// TwinCAT 3 PLC project DAS_CoreSys
// Title: DAS_TaiXin
// Company: Jidain
// ProjectVersion: 1.0.1
// ProgramVersion: 3.1.4026.20
// libraries:
//   AxisInterface_Type03, * (Beckhoff Automation)
//   BATW_Base, * (Beckhoff Automation)
//   Common Behaviour Model, * (3S - Smart Software Solutions GmbH)
//   Tc2_EtherCAT, * (Beckhoff Automation GmbH)
//   Tc2_Math, * (Beckhoff Automation GmbH)
//   Tc2_ModbusRTU, * (Beckhoff Automation GmbH)
//   Tc2_SerialCom, * (Beckhoff Automation GmbH)
//   Tc2_Standard, * (Beckhoff Automation GmbH)
//   Tc2_System, * (Beckhoff Automation GmbH)
//   Tc2_Utilities, * (Beckhoff Automation GmbH)
//   Tc3_JsonXml, * (Beckhoff Automation GmbH)
//   Tc3_MC2_AdvancedHoming, * (Beckhoff Automation GmbH)
//   Tc3_Module, * (Beckhoff Automation GmbH)
//   Tc3_PackML_V2, * (Beckhoff Automation GmbH)
//   Util, * (System)
// project tree:
//   / CoreSys.TcTTO (not stored), ModbusTask.TcTTO, MotionSync.TcTTO (not stored)
//   Library/00_PackML/01_ObjectBase/ eModeChangeState.TcDUT (not stored), FB_ModeBase_V1.TcPOU (not stored), FB_ModeBase_V2.TcPOU, I_ErrorElement.TcIO (not stored), I_ErrorSubject.TcIO (not stored)
//   Library/00_PackML/02_Mode/ E_Severity.TcDUT (not stored), E_UnitMode.TcDUT
//   Library/10_Machine/00_BaseFBs/01_FB_ObjectBase/DUTs/ E_MethodStatus_Basic.TcDUT (not stored), ST_CmdContent.TcDUT (not stored), ST_MsgContent.TcDUT (not stored)
//   Library/10_Machine/00_BaseFBs/01_FB_ObjectBase/ FB_ObjectBase.TcPOU (not stored), FB_ObjectBase_V2.TcPOU
//   Library/10_Machine/00_BaseFBs/01_FB_ObjectBase/GVLs/ Para_ObjectBase.TcGVL (not stored)
//   Library/10_Machine/00_BaseFBs/01_FB_ObjectBase/ITFs/ IBasicElement.TcIO (not stored)
//   Library/10_Machine/11_IOData/ GVL_EIP.TcGVL (not stored), GVL_Input.TcGVL (not stored), GVL_Output.TcGVL (not stored)
//   Library/10_Machine/12_MachineControl/DUTs/ AxisNo.TcDUT (not stored), E_DataFrom.TcDUT (not stored), ST_ChangeIntoProduction.TcDUT (not stored), ST_CylinderMonitor.TcDUT (not stored), ST_MotorMonitor.TcDUT (not stored), ST_TableMoveCtrl.TcDUT (not stored), ST_TableMoveService.TcDUT (not stored), ST_TableMoveStatus.TcDUT (not stored), UnitNo.TcDUT (not stored)
//   Library/10_Machine/12_MachineControl/DUTs/Cylinders/ ST_CylinderList.TcDUT, UNI_CylinderList.TcDUT (not stored)
//   Library/10_Machine/12_MachineControl/DUTs/FanucRobot/ ST_FanucRobotList.TcDUT, UNI_FanucRobotList.TcDUT
//   Library/10_Machine/12_MachineControl/DUTs/Motor/ ST_MotorList.TcDUT (not stored), UNI_MotorList.TcDUT (not stored), ST_SameSizeCVRequest.TcDUT
//   Library/10_Machine/12_MachineControl/DUTs/Service/ ST_ServiceCtrl_Base.TcDUT (not stored), ST_ServiceStatus_Base.TcDUT (not stored)
//   Library/10_Machine/12_MachineControl/DUTs/Setup/ E_ClipNo.TcDUT (not stored), ST_AllocateRobotCoordinate.TcDUT (not stored), ST_AllocateRobotPositionTable.TcDUT (not stored), ST_AxisPara.TcDUT, ST_AxisPara_Auto.TcDUT (not stored), ST_AxisPara_HalfAuto.TcDUT (not stored), ST_AxisPara_Homing.TcDUT (not stored), ST_AxisPara_Manual.TcDUT (not stored), ST_CylinderPara.TcDUT (not stored), ST_FanucRobotCCDSetting.TcDUT (not stored), ST_OutRobotCoordinate.TcDUT (not stored), ST_OutRobotPositionTable.TcDUT (not stored), ST_PositionTable.TcDUT, ST_SetupAxis.TcDUT, ST_SetupCylinder.TcDUT (not stored), ST_SetupFanucRobot.TcDUT, ST_SetupMotor.TcDUT, ST_SetupPara.TcDUT, ST_Setup_Light.TcDUT, ST_Setup_Mechanical.TcDUT
//   Library/10_Machine/12_MachineControl/ FB_MachineControl.TcPOU, GVL_Machine.TcGVL, GVL_Machine_Const.TcGVL
//   Library/10_Machine/12_MachineControl/Service/ FB_BuzzCtrl.TcPOU, FB_MachineHoming.TcPOU, FB_MachineModeSwitch.TcPOU
//   Library/10_Machine/13_ErrorHandling/ FB_ErrorHandler.TcPOU (not stored), FB_ErrorHandler_V2.TcPOU, GVL_ErrorCode.TcGVL
//   Library/10_Machine/18_HMI_Handshake/DUTs/Allocated/ ST_Auto_Allocated.TcDUT (not stored), ST_AXIS_HOMING.TcDUT (not stored), ST_AXIS_JOG.TcDUT (not stored), ST_AXIS_PTP.TcDUT (not stored), ST_HalfAuto_Allocated.TcDUT (not stored), ST_HMI_AllocateArea.TcDUT, ST_Manual_Allocated.TcDUT, ST_Manual_AllocatedRobot.TcDUT, ST_Manual_Axis.TcDUT, ST_Manual_OutRobot.TcDUT (not stored), ST_Manual_PullOut.TcDUT, ST_Manual_RoundBelt.TcDUT, ST_Manual_TransCV.TcDUT, ST_Manual_TurnTable.TcDUT (not stored)
//   Library/10_Machine/18_HMI_Handshake/DUTs/Component/ ST_DoubleValve.TcDUT (not stored), ST_MotorCommand.TcDUT (not stored), ST_SignleValve.TcDUT (not stored)
//   Library/10_Machine/18_HMI_Handshake/DUTs/ E_AllocationJob.TcDUT
//   Library/10_Machine/18_HMI_Handshake/DUTs/IOMonitor/ ST_HMI_IOMonitor.TcDUT, ST_InputTable_MitsubishiWithWheelHouse.TcDUT, ST_Input_IOMonitor.TcDUT (not stored), ST_Output_IOMonitor.TcDUT (not stored), ST_WheelhouseInput.TcDUT (not stored), ST_WheelhouseTour.TcDUT (not stored), ST_Wheelhouse_Layer.TcDUT (not stored), UNI_HMI_WheelHouseInput.TcDUT (not stored), UNI_HMI_WheelHouseInput2.TcDUT (not stored) (excluded from build)
//   Library/10_Machine/18_HMI_Handshake/DUTs/Shipping/ ST_Auto_Shipping.TcDUT (not stored), ST_HalfAuto_Shipping.TcDUT (not stored), ST_HMI_ShippingArea.TcDUT, ST_Manual_Shipping.TcDUT (not stored)
//   Library/10_Machine/18_HMI_Handshake/DUTs/Status/ ST_AllocateStatus.TcDUT (not stored), ST_Auto_Status.TcDUT (not stored), ST_AXES_STATUS.TcDUT, ST_MotorStatus.TcDUT (not stored), ST_SINGLEAXIS_STATUS.TcDUT (not stored), ST_CylinderStatus.TcDUT (not stored), ST_HalfAuto_Status.TcDUT (not stored), ST_HMI_MachineStatus.TcDUT, ST_Manual_Status.TcDUT (not stored), ST_ShippingStatus.TcDUT (not stored), ST_StorageStatus.TcDUT (not stored)
//   Library/10_Machine/18_HMI_Handshake/DUTs/Storage/ ST_Auto_Storage.TcDUT (not stored), ST_HalfAuto_Storage.TcDUT (not stored), ST_HMI_StorageArea.TcDUT, ST_Manual_FanucRobot.TcDUT, ST_Manual_Rack.TcDUT (not stored), ST_Manual_UpCV.TcDUT (not stored), ST_Manual_LowCV.TcDUT (not stored), ST_Manual_Storage.TcDUT (not stored)
//   Library/10_Machine/18_HMI_Handshake/ FB_HmiHandShake.TcPOU, GVL_ADS.TcGVL, GVL_HMI.TcGVL
//   Library/10_Machine/18_HMI_Handshake/OLD_DUTs/ E_FeedInToWareHouse_PlaceArea.TcDUT, ST_AutoMode_FeedInToWareHouseBox.TcDUT, ST_AutoMode_RobotSelfHoming.TcDUT, ST_AutoMode_ShippingLeftSideTransCV.TcDUT, E_ClampWork.TcDUT, E_FeedInEmptyBox_PickUpArea.TcDUT, E_FeedInEmptyBox_PlaceArea.TcDUT, E_HoleIndex_X.TcDUT, E_HoleIndex_Y.TcDUT, E_MachineMode.TcDUT, E_MachineState.TcDUT, E_PullOutConveyorAddress.TcDUT, E_PullOutConveyorCommandType.TcDUT, E_PullOutConveyorState.TcDUT, E_RackState.TcDUT, E_ReloadRoundBelt_PickupArea.TcDUT, E_ReloadRoundBelt_PlaceAddress.TcDUT, E_ReloadRoundBelt_PlaceArea.TcDUT, E_RobotArea.TcDUT, E_RobotClamp.TcDUT, E_RoundBeltStation.TcDUT, E_SimpleAllocateTable.TcDUT, E_WareHouse.TcDUT, E_WareHouseLayer.TcDUT, E_WareHouseSlide.TcDUT, stPositionCommand.TcDUT, st_ads_AllocateMoveStructure.TcDUT, st_ads_MachineReset.TcDUT, st_ads_OneAxisMoveWithoutPosition.TcDUT, st_ads_OneAxisMoveWithPosition.TcDUT, st_ads_OutRobtToPlateMove.TcDUT, st_ads_RobotToAllocateMove.TcDUT, ST_Alarm_Tmax.TcDUT, st_AllocateCircleMoveStructure.TcDUT, st_AllocateRobotNeedlingMove.TcDUT, ST_AllocateRobotNeedlingMoveInfo.TcDUT, st_AllocatingNeedleInfo.TcDUT, ST_AllocationJobBatchMode.TcDUT, ST_AllocationJobBatchModeInfo.TcDUT, ST_AllocationJobBatchMode_1.TcDUT, ST_AutoAddsBoxes.TcDUT, ST_AutoAddsBoxesCommand.TcDUT, ST_AutoAddsBoxesStatus.TcDUT, st_AutoMode_AllocatingJob.TcDUT, st_AutoMode_AllocatingJob_1.TcDUT, st_AutoMode_ClampingBoxesJob.TcDUT, st_AutoMode_ClampingToPlate.TcDUT, ST_AutoMode_DetectDiameter.TcDUT, ST_AutoMode_FeedInEmptyBox.TcDUT, ST_AutoMode_ReloadRoundBeltBox.TcDUT, ST_AutoMode_RobotRegionMove.TcDUT, ST_AutoMode_ShippingLeftSideTransCVFeedBack.TcDUT, ST_AutoMode_ShippingLeftSideTransCVInfo.TcDUT, ST_AutoMode_ShippingRightSideTransCV.TcDUT, ST_AutoMode_SimpleAllocateHandShake.TcDUT, st_AutoMode_SingleStepWithInterventionRequest.TcDUT, ST_AutoMode_TransCVCamera.TcDUT, ST_AutoMode_WareHouseInnerPickToRoundBelt.TcDUT, E_ShippingPlateIndex.TcDUT, E_ShippingPlateSide.TcDUT, ST_ShippingPlateToConveyor.TcDUT, ST_AutoPullOutConveyor.TcDUT, ST_AutoPullOutConveyorCommand.TcDUT, ST_AutoPullOutConveyorSatus.TcDUT, ST_AutoServoPara.TcDUT, st_AutoSixAxisAbsMoveParameter.TcDUT, st_AutoSixAxisWarehouseParameter.TcDUT, st_AutoSperate.TcDUT, ST_Auto_LowerFeedInConveyor.TcDUT, ST_Auto_LowerFeedInConveyorCommand.TcDUT, ST_Auto_LowerFeedInConveyorStatus.TcDUT, ST_Auto_UpperFeedInConveyor.TcDUT, ST_Auto_UpperFeedInConveyorCommand.TcDUT, ST_Auto_UpperFeedInConveyorFeedback.TcDUT, ST_Auto_UpperFeedInConveyorInfo.TcDUT, ST_Auto_UpperFeedInConveyorStatus.TcDUT, st_AxisControl.TcDUT, ST_BuzzCtrl.TcDUT, ST_ClampActionRecord.TcDUT, st_ClampingBoxesInfo.TcDUT, ST_ClampSetting.TcDUT, ST_ClampSetting_FeedInToWareHouse.TcDUT, ST_ClampSetting_ReloadRoundBelt.TcDUT, ST_CommandBasic.TcDUT, ST_DetectDiameterCommand.TcDUT, ST_DetectDiameterInfo.TcDUT, ST_DetectDiameterStatus.TcDUT, ST_FanucRobotGeneralCtrl.TcDUT, ST_FanucRobotReadAllOffssetDate.TcDUT, ST_FanucRobotReadSingleOffsetData.TcDUT, ST_FanucRobotWriteAllOffsetDate.TcDUT, ST_FanucRobotWriteSingleOffsetData.TcDUT, ST_FanucRobot_CSharpCommand.TcDUT, ST_FanucRobot_CSharpStatus.TcDUT, ST_FeedInEmptyBox_Ctrl.TcDUT, ST_FeedInEmptyBox_Info.TcDUT, ST_FeedInEmptyBox_Status.TcDUT, ST_FeedInRBActionRecord.TcDUT, ST_FeedInRBBatch.TcDUT, ST_FeedInRBFlowInfo.TcDUT, ST_FeedInToWareHouseBox_Info.TcDUT, ST_FeedInToWareHouse_Ctrl.TcDUT, ST_FeedInToWareHouse_Status.TcDUT, st_FlowBaseCore.TcDUT, st_HandshakeBase.TcDUT, st_HandShakeBaseWithError.TcDUT, st_ListRunCore.TcDUT, ST_ManualServoPara.TcDUT, ST_MechanicalList.TcDUT, st_ModbusSwitchOff.TcDUT, ST_Mode.TcDUT, st_MoveConveyorJob.TcDUT, ST_OffsetData.TcDUT, st_OneDirectionCore.TcDUT, ST_OneProcessServoPara.TcDUT, ST_OpPannelStatus.TcDUT, st_OutRobotParameterCore.TcDUT, ST_PositionOffsetData.TcDUT, ST_PullOutConveyorInfo.TcDUT, ST_ReadAllOffsetDataCommand.TcDUT, ST_ReadAllOffsetDateStatus.TcDUT, ST_ReadSingleOffsetData_Command.TcDUT, ST_ReadSingleOffsetData_Info.TcDUT, ST_ReadSingleOffsetData_Status.TcDUT, st_RegionHome.TcDUT (not stored), ST_ReloadRoundBeltBox_Info.TcDUT, ST_ReloadRoundBelt_Ctrl.TcDUT, ST_ReloadRoundBelt_Status.TcDUT, st_Robot.TcDUT, st_RobotMoveAbs.TcDUT, ST_RobotRegionMove_Info.TcDUT, ST_RoundBeltCoordinates.TcDUT, st_SafetyByPass.TcDUT, ST_SaveParaDefault.TcDUT, ST_SaveParaRemote.TcDUT, st_ServiceTimeoutSetting.TcDUT, ST_ServoList.TcDUT, ST_ServoParaBasic.TcDUT, ST_SimpleAllocateCommand.TcDUT, ST_SimpleAllocateInfo.TcDUT, ST_SimpleAllocateStatus.TcDUT, st_SixAxisRobotCore.TcDUT, st_SixAxisWarehouseParameter.TcDUT, st_StationPositions.TcDUT, ST_StatusBasic.TcDUT, ST_SystemParameter.TcDUT, ST_WareHouseCoordinates.TcDUT, ST_WareHouseInnerPickBatch.TcDUT, ST_WareHouseInnerPickFlowInfo.TcDUT, ST_WriteAllOffsetData_Command.TcDUT, ST_WriteAllOffsetData_Info.TcDUT, ST_WriteAllOffsetData_Status.TcDUT, ST_WriteSingleOffsetData_Command.TcDUT, ST_WriteSingleOffsetData_Info.TcDUT, ST_WriteSingleOffsetData_Status.TcDUT
//   Library/10_Machine/18_HMI_Handshake/OLD_DUTs/DataCore/ st_ADSBaseParaCore.TcDUT (not stored), st_ADSMotoCore.TcDUT (not stored), st_ADSMotoMoveCore.TcDUT (not stored), st_ADS_X.TcDUT, st_ADS_Y.TcDUT, st_AllocateParameterCore.TcDUT (not stored), st_DASCalibrationData.TcDUT (not stored)
//   Library/10_Machine/18_HMI_Handshake/Service/DUTs/AllocateBatchMode/ st_AllocateMoveAutoBatchMode_Ctrl.TcDUT (not stored), st_AllocateMoveAutoBatchMode_Status.TcDUT (not stored), st_Coordinate.TcDUT (not stored), ST_Cylinders.TcDUT (not stored), st_RoundBeltAutoSingleMove_Ctrl.TcDUT (not stored), U_Cylinders.TcDUT (not stored)
//   Library/10_Machine/18_HMI_Handshake/Service/DUTs/ ST_HMI_Handshake.TcDUT
//   Library/10_Machine/19_Device/EL1889/ ST_EbusDI16.TcDUT (not stored), ST_EbusInputModule.TcDUT (not stored), ST_InputTable.TcDUT, ST_InputTable_Mitsubishi.TcDUT (not stored), uni_InputModule.TcDUT (not stored)
//   Library/10_Machine/19_Device/EL2889/ ST_EbusDO16.TcDUT (not stored), ST_EbusOutputModule.TcDUT (not stored), ST_OutputTable.TcDUT, ST_OutputTable_Mitsubishi.TcDUT, uni_OutputModule.TcDUT
//   Library/10_Machine/19_Device/FanucRobot/DUTs/ E_ClampAction.TcDUT (not stored), E_FanucRobotOpMode.TcDUT (not stored), E_PullOutConveyorPosition.TcDUT (not stored), E_RobotAddress.TcDUT (not stored), ST_AutoMode_ShippingRobotTransfer.TcDUT, ST_AutoMode_ShippingRobot_MoveAbs.TcDUT, ST_CCD_ZoneUse.TcDUT (not stored), ST_FanucUI1.TcDUT (not stored), ST_FanucUO1.TcDUT (not stored), ST_Fanuc_AbsMove.TcDUT (not stored), ST_Fanuc_GeneralCommand.TcDUT (not stored), ST_Fanuc_GeneralCommand_1.TcDUT (not stored), ST_Fanuc_Status.TcDUT (not stored), ST_Fanuc_WarehouseHandshake.TcDUT (not stored), ST_IntToBool.TcDUT (not stored), ST_ReadWriteParaCmd.TcDUT (not stored), ST_ReadWriteParaStatus.TcDUT
//   Library/10_Machine/19_Device/FanucRobot/ FB_FanucRobot_Basic.TcPOU (excluded from build), FB_FanucRobot_Basic_V2.TcPOU (unreadable)
//   Library/20_MachineUnits/21_StorageArea/210_Cabinet/DUTs/ E_CabinetJob.TcDUT (not stored), st_LayerStatus.TcDUT (not stored), st_WarehouseLayer.TcDUT (not stored), st_WarehouseList.TcDUT (not stored), U_Bits_To_stStatus.TcDUT (not stored), _st_LayerStatus.TcDUT (not stored), _st_WareHouseLayer.TcDUT (not stored), _st_WarehouseList.TcDUT (not stored)
//   Library/20_MachineUnits/21_StorageArea/210_Cabinet/ FB_WareHouse.TcPOU
//   Library/20_MachineUnits/21_StorageArea/210_Cabinet/Services/ FB_FeedInBox.TcPOU, FB_ReloadBox.TcPOU
//   Library/20_MachineUnits/21_StorageArea/Duts/ E_FeedInAction.TcDUT (not stored), E_FeedInToWareHouseAction.TcDUT, E_ReloadRoundBoxAction.TcDUT (not stored), st_RebootModbusDevices.TcDUT, st_RobotAbsMove_Ctrl.TcDUT (not stored), st_RobotAbsMove_Status.TcDUT (not stored), st_RobotWarehouseMove_Ctrl.TcDUT (not stored), st_RobotWarehouseMove_Status.TcDUT (not stored), ST_StorageService.TcDUT
//   Library/20_MachineUnits/21_StorageArea/ FB_StorageArea.TcPOU
//   Library/20_MachineUnits/21_StorageArea/Old_version_Service/ FB_FeedInEmptyBoxWithRobot.TcPOU (excluded from build), FB_FeedInEmptyBoxWithRobot_V2.TcPOU (not stored) (excluded from build), FB_FeedInEmptyBoxWithRobot_V3.TcPOU, FB_FeedInRoundBeltBoxBatch_Old.TcPOU (excluded from build), FB_FeedInRoundBeltBoxToWareHouse_Old.TcPOU (excluded from build), FB_FeedInRoundBeltBoxToWareHouse_OldV2.TcPOU (excluded from build), FB_ReloadRoundBeltBoxWithRobot.TcPOU (not stored) (excluded from build), FB_RobotAbsMove.TcPOU (excluded from build), FB_RobotRegionMove_FeedInConveyor.TcPOU (excluded from build), FB_WareHouseInnerPickToRoundBeltBatch_Old.TcPOU (excluded from build), FB_WareHouseWithRobotMove.TcPOU (not stored) (excluded from build)
//   Library/20_MachineUnits/21_StorageArea/Service/ FB_AddBoxes_v2.TcPOU, FB_BoxSupplyCtrl.TcPOU, FB_BoxSupplyCtrl_v1.TcPOU, FB_DiameterMovement.TcPOU, FB_LowerFeedInConveyor.TcPOU, FB_RebootModbusDevice.TcPOU, FB_StorageHoming.TcPOU, FB_UpperFeedInConveyor.TcPOU
//   Library/20_MachineUnits/21_StorageArea/Service_Robot/ FB_FeedInEmptyBoxWithRobot_V4.TcPOU, FB_FeedInRoundBeltBoxBatch.TcPOU, FB_FeedInRoundBeltBoxToWareHouse.TcPOU, FB_ReloadRoundBeltBoxWithRobot_V2.TcPOU, FB_RobotAbsMove_V2.TcPOU, FB_RobotRegionMove_AllocatedConveyor.TcPOU, FB_RobotRegionMove_BufferArea.TcPOU, FB_RobotRegionMove_FeedInConveyor_V2.TcPOU, FB_RobotRegionMove_PullOutConveyor.TcPOU, FB_RobotRegionMove_RoundBelt.TcPOU, FB_RobotSelfHoming.TcPOU, FB_WareHouseInnerPickToRoundBelt.TcPOU, FB_WareHouseInnerPickToRoundBeltBatch.TcPOU, FB_WareHouseWithRobotMove_V3.TcPOU
//   Library/20_MachineUnits/22_AllocateArea/Duts/Enums/ E_RoundBeltControlAccess.TcDUT (not stored)
//   Library/20_MachineUnits/22_AllocateArea/Duts/ E_Pistons.TcDUT (not stored), F_Even.TcPOU (not stored), ST_AllocateService.TcDUT, ST_AutoMode_ReverseBatchPick.TcDUT, E_ReverseBoxDestination.TcDUT, ST_AutoMode_ReverseBoxToWareHouse.TcDUT, ST_DuoCylinders.TcDUT (not stored), ST_ReverseBatchBoxQueue.TcDUT, ST_ReverseBatchBoxResult.TcDUT, st_RoundBeltAutoSingleMove_Status.TcDUT (not stored), Uni_DuoCylinders.TcDUT (not stored)
//   Library/20_MachineUnits/22_AllocateArea/ FB_AllocateAreaWithRoundbelt.TcPOU, FB_AllocateAreaWithXPlanar.TcPOU (not stored)
//   Library/20_MachineUnits/22_AllocateArea/FUNs/ FUN_GetNeedleCoordinates.TcPOU (not stored), FUN_GetSyncGroup_AllocationJob.TcPOU (not stored)
//   Library/20_MachineUnits/22_AllocateArea/Old_Version_Service/ FB_AllocateMoveAutoBatchMode_Reverse_Old.TcPOU (excluded from build), FB_OutRobot_BoxMoveReverse_Old.TcPOU (excluded from build), FB_OutRobot_EmptyBoxMove_old.TcPOU (excluded from build), FB_OutRobot_RareBoxMove_old.TcPOU (excluded from build), FB_PullOutConveyorAction_OLD.TcPOU (excluded from build), FB_PullOutConveyorBtnCtrl_OLD.TcPOU (excluded from build)
//   Library/20_MachineUnits/22_AllocateArea/Service/ FB_AllocateMoveAutoBatchMode_Reverse.TcPOU, FB_AllocateRobotNeedlingMove.TcPOU, FB_AllocateMoveAutoBatchMode.TcPOU, FB_OutRobot_BoxMoveReverse.TcPOU, FB_OutRobot_EmptyBoxMove.TcPOU, FB_OutRobot_BoxMoveTurnTableToRoundBelt.TcPOU, FB_OutRobot_RareBoxMove.TcPOU, FB_PullOutConveyorAction.TcPOU, FB_PullOutConveyorBtnCtrl.TcPOU (not stored), FB_RoundBeltService.TcPOU, FB_AllocateAreaHome.TcPOU, FB_SameSizeCVCamera.TcPOU, FB_DifferentCVCamera.TcPOU, FB_SameSizeCVCamera_Reverse.TcPOU, FB_SameSizeCV_ReverseBatchPickAndPhoto.TcPOU, FB_SameSizeCV_ReverseBoxToWareHouse.TcPOU, FB_TurnTableService.TcPOU
//   Library/20_MachineUnits/23_ShippingArea/Duts/ ST_BlinkInfo.TcDUT, ST_ShippingRobotTransfer_AreaInfo.TcDUT, ST_ShippingRobotTransfer_Info.TcDUT, ST_ShippingService.TcDUT
//   Library/20_MachineUnits/23_ShippingArea/ FB_ShippingArea.TcPOU, FB_ShippingHoming.TcPOU
//   Library/20_MachineUnits/23_ShippingArea/RobotService/ FB_ShippingRobotTransfer.TcPOU, FB_ShippingRobot_Buffer.TcPOU, FB_ShippingPlateScan.TcPOU, FB_ShippingRobot_Left.TcPOU, FB_ShippingRobot_PhotoStandByPos.TcPOU, FB_ShippingRobot_Right.TcPOU, FB_ShippingRobot_TransmitCVEnd.TcPOU
//   Library/20_MachineUnits/23_ShippingArea/Service/ FB_ShippingTransCV_LeftSide.TcPOU, FB_ShippingTransCV_RightSide.TcPOU
//   Library/99_Utilities/Duts/ E_SignalTowerLampMode.TcDUT (not stored), ST_BoolList.TcDUT (not stored), ST_SignalTower.TcDUT (not stored), uni_IntToBool.TcDUT (not stored)
//   Library/99_Utilities/ErrorHandling/ FB_ErrorHandler_OLD.TcPOU (not stored) (excluded from build), FB_ErrorHandler_abond.TcPOU (not stored) (excluded from build), FB_ErrorHandling.TcPOU (not stored) (excluded from build)
//   Library/99_Utilities/ FB_CylinderManualCtrl.TcPOU, FB_EdgeDetect.TcPOU (not stored), FB_MotorManualCtrl.TcPOU, FB_SignalGen.TcPOU (not stored), FB_SignalTower.TcPOU, FB_TableMove.TcPOU, FB_XY_Move.TcPOU (not stored), FB_XY_PickAndPlace.TcPOU (not stored), F_FtoPT.TcPOU (not stored)
//   Library/99_Utilities/FUNCTION/ FUN_CheckAxisAllowMove.TcPOU (not stored), FUN_CheckInPos.TcPOU, FUN_GetPositionTableData.TcPOU (not stored), FUN_MachineState.TcPOU (not stored), FUN_ResetStorageCylinder.TcPOU (not stored), FUN_RetractStorageCylinder.TcPOU (not stored)
//   Library/30_Simulation/ GVL_SimMode.TcGVL
//   Library/30_Simulation/10_IOSim/ FB_SimulatedIO.TcPOU
//   POUs/CheckProg/ CheckBounds.TcPOU (not stored), CheckDivDInt.TcPOU (not stored), CheckDivLInt.TcPOU (not stored), CheckDivLReal.TcPOU (not stored), CheckDivReal.TcPOU (not stored), CheckLRangeSigned.TcPOU (not stored), CheckLRangeUnsigned.TcPOU (not stored), CheckPointer.TcPOU (not stored), CheckRangeSigned.TcPOU (not stored), CheckRangeUnsigned.TcPOU (not stored)
//   POUs/ DAS_CoreSys.TcPOU, DAS_MotionSync.TcPOU (not stored)
//   POUs/ModbusRTU/00_BaseFBs/01_FB_ObjectBase/ FB_ObjectBase_V2.TcPOU (not stored)
//   POUs/ModbusRTU/ ComModbusRTU.TcPOU
//   POUs/ModbusRTU/SerialComTask/DUTs/ un_RS485States.TcDUT (not stored), un_RS485States_all.TcDUT (not stored)
//   POUs/ModbusRTU/SerialComTask/ FB_CommunicateModbusRTU.TcPOU
//   POUs/RS485_JidianVersion/DUTs/ ST_RS485Controller.TcDUT, ST_RS485_Heartbeat.TcDUT, ST_RS485_LayerStatus.TcDUT, ST_RS485_SliderStatusALL.TcDUT
//   POUs/RS485_JidianVersion/ FB_WarehouseSensorCtrl.TcPOU, MAIN2_RS485.TcPOU
// real-time tasks:
//   TASK CoreSys: cycle T#10ms, priority 20, ADS port 350
//   TASK MotionSync: cycle T#2ms, priority 1, ADS port 351
//   TASK EIP_Task: cycle T#2ms, priority 2, ADS port 301
//   TASK ModbusTask: cycle T#5ms, priority 21, ADS port 352
// motion (NC):
//   TASK NC-Task 1 SAF: cycle T#2ms, priority 4, ADS port 501
//   TASK NC-Task 1 SVB: cycle T#2ms, priority 8, ADS port 511
//   AXIS Axis 1|TurnTable (id 1)
//     General: UnitName=°
//     Dynamic: Acceleration=1800, Deceleration=1800, Jerk=10800
//     Velo: SlowManual=6, FastManual=60, Maximum=600
//     OtherSettings: AllowMotionCmdToSlave=true
//     encoder EncType=19
//       EncPara: ScaleFactorNumerator=120, ScaleFactorDenominator=83886080, MaxCount=#xffffffff
//         SoftEndMaxControl: Range=350
//         Inc: RefSoftSyncMask=#x0000ffff
//     drive DrvType=16
//       DrvPara: MaxCount=#xffffffff, DriveControlDWord=#x00020100
//         Analog: VeloReferenz=600, TorqueSetpointScale=10, ScaleFactorActTorque=0.1
//         TimeComp: TaskDelayCycles=1
//     controller CtrType=1
//       CtrPara: PriorControlFactor=1
//         PosDiffControl: Enable=false
//         Observer: BandWidth=20
//   AXIS Axis 2|RoundBelt (id 2)
//     General: UnitFlags=#x00000004
//     Dynamic: AccelerationMaximum=3900, DecelerationMaximum=3900, Acceleration=3900, Deceleration=3900, Jerk=30000
//     Velo: SlowManual=6, FastManual=200, Maximum=500
//     OtherSettings: AllowMotionCmdToSlave=true
//     encoder EncType=19
//       EncPara: ScaleFactorNumerator=500, ScaleFactorDenominator=167772160, ModuloFactor=2800, MaxCount=#xffffffff
//         Inc: RefSoftSyncMask=#x0000ffff
//     drive DrvType=16
//       DrvPara: MaxCount=#xffffffff, DriveControlDWord=#x00020100
//         Analog: VeloReferenz=500, TorqueSetpointScale=10, ScaleFactorActTorque=0.1
//         TimeComp: TaskDelayCycles=1
//     controller CtrType=1
//       CtrPara: PriorControlFactor=1
//         PosDiffControl: Range=10
//         Observer: BandWidth=20
//   AXIS Axis 3|AllocateRobot_X (id 3)
//     Dynamic: Acceleration=12000, Deceleration=12000, Jerk=360000
//     Velo: SlowManual=6, FastManual=60, Maximum=800
//     OtherSettings: AllowMotionCmdToSlave=true
//     encoder EncType=19
//       EncPara: ScaleFactorNumerator=36, ScaleFactorDenominator=8388608, MaxCount=#xffffffff
//         Inc: RefSoftSyncMask=#x0000ffff
//     drive DrvType=16
//       DrvPara: MaxCount=#xffffffff, DriveControlDWord=#x00020100
//         Analog: TorqueSetpointScale=10, ScaleFactorActTorque=0.1
//         TimeComp: TaskDelayCycles=1
//     controller CtrType=1
//       CtrPara: PriorControlFactor=1
//         Observer: BandWidth=20
//   AXIS Axis 4|AllocateRobot_Y (id 4)
//     Dynamic: Acceleration=15000, Deceleration=15000, Jerk=225000
//     OtherSettings: AllowMotionCmdToSlave=true
//     encoder EncType=19
//       EncPara: ScaleFactorNumerator=16, ScaleFactorDenominator=8388608, Inverse=true, MaxCount=#xffffffff
//         Inc: RefSoftSyncMask=#x0000ffff
//     drive DrvType=16
//       DrvPara: Inverse=true, MaxCount=#xffffffff, DriveControlDWord=#x00020100
//         Analog: TorqueSetpointScale=10, ScaleFactorActTorque=0.1
//         TimeComp: TaskDelayCycles=1
//     controller CtrType=1
//       CtrPara: PriorControlFactor=1
//         PosDiffControl: Range=10
//         Observer: BandWidth=20
//   AXIS Axis 5|OutRobot_X (id 5)
//     Dynamic: Acceleration=11250, Deceleration=11250, Jerk=168750
//     Velo: SlowManual=6, FastManual=60, Maximum=1500
//     OtherSettings: AllowMotionCmdToSlave=true
//     encoder EncType=19
//       EncPara: ScaleFactorNumerator=30, ScaleFactorDenominator=8388608, MaxCount=#xffffffff
//     drive DrvType=16
//       DrvPara: MaxCount=#xffffffff, DriveControlDWord=#x00020100
//         Analog: TorqueSetpointScale=10, ScaleFactorActTorque=0.1
//         TimeComp: TaskDelayCycles=1
//     controller CtrType=1
//       CtrPara: PriorControlFactor=1
//         PosDiffControl: Range=10
//         Observer: BandWidth=20
//   AXIS Axis 6|OutRobot_Y (id 6)
//     Dynamic: Acceleration=6000, Deceleration=6000, Jerk=36000
//     Velo: SlowManual=6, FastManual=60
//     OtherSettings: AllowMotionCmdToSlave=true
//     encoder EncType=19
//       EncPara: ScaleFactorNumerator=40, ScaleFactorDenominator=8388608, MaxCount=#xffffffff
//     drive DrvType=16
//       DrvPara: MaxCount=#xffffffff, DriveControlDWord=#x00020100
//         Analog: TorqueSetpointScale=10, ScaleFactorActTorque=0.1
//         TimeComp: TaskDelayCycles=1
//     controller CtrType=1
//       CtrPara: PriorControlFactor=1
//         PosDiffControl: Range=10
//         Observer: BandWidth=20
//   AXIS Axis 7|RackMotor (id 7)
//     Dynamic: Acceleration=800.624, Deceleration=800.624, Jerk=1167.58
//     Velo: SlowManual=5, FastManual=100, Maximum=732
//     OtherSettings: AllowMotionCmdToSlave=true
//     encoder EncType=4
//       EncPara: ScaleFactorNumerator=90, ScaleFactorDenominator=980, MaxCount=#xffffffff
//     drive DrvType=23
//       Analog: VeloReferenz=732, TorqueSetpointScale=10, ScaleFactorActTorque=0.1
//       TimeComp: TaskDelayCycles=1
//     controller CtrType=1
//       CtrPara: PriorControlFactor=1
//         PID: PosKp=90
//         Observer: BandWidth=20
// I/O:
//   DEVICE Device 1 (EtherCAT) Storage, AmsNetId 169.254.53.69.2.1
//     Term 1 (EK1200) [EK1200-5000 EtherCAT Power supply (2A E-Bus)]
//       Term 2 (EL6021) [EL6021 Interface (RS422/485)]
//       Term 3 (EL6021) [EL6021 Interface (RS422/485)]
//       Term 4 (EL6021) [EL6021 Interface (RS422/485)]
//       Term 5 (EL6021) [EL6021 Interface (RS422/485)]
//       Term 6 (EL1889)_01(X6) [EL1889 16Ch. Dig. Input 24V, 3ms, negative]
//       Term 7 (EL1889)_02(X7) [EL1889 16Ch. Dig. Input 24V, 3ms, negative]
//       Term 8 (EL1889)_03(X9) [EL1889 16Ch. Dig. Input 24V, 3ms, negative]
//       Term 9 (EL1889)_04(X10) [EL1889 16Ch. Dig. Input 24V, 3ms, negative]
//       Term 10 (EL2889)_01(Y4) [EL2889 16Ch. Dig. Output 24V, 0.5A, negative]
//       Term 11 (EL2889)_02(Y5) [EL2889 16Ch. Dig. Output 24V, 0.5A, negative]
//       Term 12 (EL2889)_03(Y6) [EL2889 16Ch. Dig. Output 24V, 0.5A, negative]
//       Term 13 (EL2889)_04(Y7) [EL2889 16Ch. Dig. Output 24V, 0.5A, negative]
//       Term 14 (EL2889)_05(Y8) [EL2889 16Ch. Dig. Output 24V, 0.5A, negative]
//       Term 59 (EL9410) [EL9410 E-Bus Power Supplier  (Diagnostics)]
//       Term 15 (EL2889)_06(Y10) [EL2889 16Ch. Dig. Output 24V, 0.5A, negative]
//       Term 17 (EL2889)_07(Y11) [EL2889 16Ch. Dig. Output 24V, 0.5A, negative]
//       Term 18 (EL7342) [EL7342 2Ch. DC motor output stage (50V, 3.5A)]
//       Term 19 (EL6652) [EL6652 EtherNet/IP Scanner (Master)]
//       Term 20 (EL9011) [EL9011 End Terminal]
//   DEVICE Device 4 (EtherCAT) Allocate, AmsNetId 169.254.53.69.5.1
//     Box 21 (CU2508) [CU2508 Ethernet Port]
//     Term 22 (EK1100) [EK1100 EtherCAT Coupler (2A E-Bus)]
//       Term 23 (EL1889)_05(X0) [EL1889 16Ch. Dig. Input 24V, 3ms, negative]
//       Term 24 (EL1889)_06(X1) [EL1889 16Ch. Dig. Input 24V, 3ms, negative]
//       Term 25 (EL1889)_07(X2) [EL1889 16Ch. Dig. Input 24V, 3ms, negative]
//       Term 26 (EL1889)_08(X3) [EL1889 16Ch. Dig. Input 24V, 3ms, negative]
//       Term 27 (EL1889)_09(X8) [EL1889 16Ch. Dig. Input 24V, 3ms, negative]
//       Term 28 (EL1889)_10(X11) [EL1889 16Ch. Dig. Input 24V, 3ms, negative]
//       Term 29 (EL2889)_08(Y0) [EL2889 16Ch. Dig. Output 24V, 0.5A, negative]
//       Term 30 (EL2889)_09(Y1) [EL2889 16Ch. Dig. Output 24V, 0.5A, negative]
//       Term 31 (EL2889)_10(Y2) [EL2889 16Ch. Dig. Output 24V, 0.5A, negative]
//       Term 32 (EL9410) [EL9410 E-Bus Power Supplier  (Diagnostics)]
//       Term 33 (EL1889)_11(X4) [EL1889 16Ch. Dig. Input 24V, 3ms, negative]
//       Term 15 (EL6652) [EL6652 EtherNet/IP Scanner (Master)]
//       Term 16 (EL9011) [EL9011 End Terminal]
//   DEVICE Device 5 (EtherCAT), AmsNetId 169.254.53.69.6.1
//     Box 37 (CU2508) [CU2508 Ethernet Port]
//     Drive 38 (MBDLT25BF) [MBDLT25BF]
//     Drive 39 (MCDLT35BF) [MCDLT35BF]
//     Drive 40 (MBDLT25BF) [MBDLT25BF]
//     Drive 41 (MADLT15BF) [MADLT15BF]
//     Drive 42 (MADLT15BF) [MADLT15BF]
//     Drive 43 (MBDLT25BF) [MBDLT25BF]
//   DEVICE Storage Fanuc Robot (ECAT EIP Scanner (EL6652)), AmsNetId 169.254.53.69.4.1
//     FANUC Robot R30iB+ // <INFO> 192.168.0.3, FANUC Robot R30iB+ (ProdCode: 4, Rev: 3.01, Mac: 00:e0:e4:c5:29:bd) </INFO> <EDS> C:\TwinCAT\3.1\Config\Io\EtherNetIP\FANUCROBOT0301_R30IBP.EDS </EDS>
//   DEVICE Device 6 (ECAT EIP Scanner (EL6652)), AmsNetId 169.254.53.69.7.1
//     FANUC Robot R30iB+ // <INFO> 192.168.0.13, FANUC Robot R30iB+ (ProdCode: 4, Rev: 3.01, Mac: 00:e0:e4:99:c3:31) </INFO> <EDS> C:\TwinCAT\3.1\Config\Io\EtherNetIP\FANUCROBOT0301_R30IBP.EDS </EDS>
//   DEVICE X001 (RT-Ethernet Adapter)
// variable links:
//   NC-Task 1 SAF/Axes/Axis 1|TurnTable <-> Device 5 (EtherCAT)/Drive 38 (MBDLT25BF)
//     Drive/Inputs/In/nDataIn1 <-> Transmit PDO mapping 1/Following error actual value
//     Drive/Inputs/In/nDcOutputTime <-> InfoData/DcOutputShift
//     Drive/Inputs/In/nState1 <-> Transmit PDO mapping 1/Statusword
//     Drive/Inputs/In/nState2 <-> Transmit PDO mapping 1/Statusword @bit 8
//     Drive/Inputs/In/nState4 @bit 1 <-> WcState/InputToggle
//     Drive/Inputs/In/nState4 <-> WcState/WcState
//     Drive/Inputs/In/nState5 <-> Transmit PDO mapping 1/Modes of operation display
//     Drive/Outputs/Out/nCtrl1 <-> Receive PDO mapping 1/Controlword
//     Drive/Outputs/Out/nCtrl2 <-> Receive PDO mapping 1/Controlword @bit 8
//     Drive/Outputs/Out/nCtrl5 <-> Receive PDO mapping 1/Modes of operation
//     Drive/Outputs/Out/nDataOut1 <-> Receive PDO mapping 1/Target position
//     Enc/Inputs/In/nDataIn1 <-> Transmit PDO mapping 1/Position actual value
//     Enc/Inputs/In/nDataIn3 <-> Transmit PDO mapping 1/Touch probe pos1 pos value
//     Enc/Inputs/In/nDcInputTime <-> InfoData/DcInputShift
//     Enc/Inputs/In/nState4 @bit 1 <-> WcState/InputToggle
//     Enc/Inputs/In/nState4 <-> WcState/WcState
//     Enc/Inputs/In/nState5 <-> Transmit PDO mapping 1/Touch probe status
//     Enc/Inputs/In/nState6 <-> Transmit PDO mapping 1/Touch probe status @bit 8
//     Enc/Outputs/Out/nCtrl5 <-> Receive PDO mapping 1/Touch probe function
//     Enc/Outputs/Out/nCtrl6 <-> Receive PDO mapping 1/Touch probe function @bit 8
//   NC-Task 1 SAF/Axes/Axis 2|RoundBelt <-> Device 5 (EtherCAT)/Drive 39 (MCDLT35BF)
//     Drive/Inputs/In/nDataIn1 <-> Transmit PDO mapping 1/Following error actual value
//     Drive/Inputs/In/nDataIn3[0] <-> Transmit PDO mapping 1/Torque actual value
//     Drive/Inputs/In/nDcOutputTime <-> InfoData/DcOutputShift
//     Drive/Inputs/In/nState1 <-> Transmit PDO mapping 1/Statusword
//     Drive/Inputs/In/nState2 <-> Transmit PDO mapping 1/Statusword @bit 8
//     Drive/Inputs/In/nState4 @bit 1 <-> WcState/InputToggle
//     Drive/Inputs/In/nState4 <-> WcState/WcState
//     Drive/Inputs/In/nState5 <-> Transmit PDO mapping 1/Modes of operation display
//     Drive/Outputs/Out/nCtrl1 <-> Receive PDO mapping 1/Controlword
//     Drive/Outputs/Out/nCtrl2 <-> Receive PDO mapping 1/Controlword @bit 8
//     Drive/Outputs/Out/nCtrl5 <-> Receive PDO mapping 1/Modes of operation
//     Drive/Outputs/Out/nDataOut1 <-> Receive PDO mapping 1/Target position
//     Enc/Inputs/In/nDataIn1 <-> Transmit PDO mapping 1/Position actual value
//     Enc/Inputs/In/nDataIn3 <-> Transmit PDO mapping 1/Touch probe pos1 pos value
//     Enc/Inputs/In/nDcInputTime <-> InfoData/DcInputShift
//     Enc/Inputs/In/nState4 @bit 1 <-> WcState/InputToggle
//     Enc/Inputs/In/nState4 <-> WcState/WcState
//     Enc/Inputs/In/nState5 <-> Transmit PDO mapping 1/Touch probe status
//     Enc/Inputs/In/nState6 <-> Transmit PDO mapping 1/Touch probe status @bit 8
//     Enc/Outputs/Out/nCtrl5 <-> Receive PDO mapping 1/Touch probe function
//     Enc/Outputs/Out/nCtrl6 <-> Receive PDO mapping 1/Touch probe function @bit 8
//   NC-Task 1 SAF/Axes/Axis 3|AllocateRobot_X <-> Device 5 (EtherCAT)/Drive 40 (MBDLT25BF)
//     Drive/Inputs/In/nDataIn1 <-> Transmit PDO mapping 1/Following error actual value
//     Drive/Inputs/In/nDcOutputTime <-> InfoData/DcOutputShift
//     Drive/Inputs/In/nState1 <-> Transmit PDO mapping 1/Statusword
//     Drive/Inputs/In/nState2 <-> Transmit PDO mapping 1/Statusword @bit 8
//     Drive/Inputs/In/nState4 @bit 1 <-> WcState/InputToggle
//     Drive/Inputs/In/nState4 <-> WcState/WcState
//     Drive/Inputs/In/nState5 <-> Transmit PDO mapping 1/Modes of operation display
//     Drive/Outputs/Out/nCtrl1 <-> Receive PDO mapping 1/Controlword
//     Drive/Outputs/Out/nCtrl2 <-> Receive PDO mapping 1/Controlword @bit 8
//     Drive/Outputs/Out/nCtrl5 <-> Receive PDO mapping 1/Modes of operation
//     Drive/Outputs/Out/nDataOut1 <-> Receive PDO mapping 1/Target position
//     Enc/Inputs/In/nDataIn1 <-> Transmit PDO mapping 1/Position actual value
//     Enc/Inputs/In/nDataIn3 <-> Transmit PDO mapping 1/Touch probe pos1 pos value
//     Enc/Inputs/In/nDcInputTime <-> InfoData/DcInputShift
//     Enc/Inputs/In/nState4 @bit 1 <-> WcState/InputToggle
//     Enc/Inputs/In/nState4 <-> WcState/WcState
//     Enc/Inputs/In/nState5 <-> Transmit PDO mapping 1/Touch probe status
//     Enc/Inputs/In/nState6 <-> Transmit PDO mapping 1/Touch probe status @bit 8
//     Enc/Outputs/Out/nCtrl5 <-> Receive PDO mapping 1/Touch probe function
//     Enc/Outputs/Out/nCtrl6 <-> Receive PDO mapping 1/Touch probe function @bit 8
//   NC-Task 1 SAF/Axes/Axis 4|AllocateRobot_Y <-> Device 5 (EtherCAT)/Drive 41 (MADLT15BF)
//     Drive/Inputs/In/nDataIn1 <-> Transmit PDO mapping 1/Following error actual value
//     Drive/Inputs/In/nDcOutputTime <-> InfoData/DcOutputShift
//     Drive/Inputs/In/nState1 <-> Transmit PDO mapping 1/Statusword
//     Drive/Inputs/In/nState2 <-> Transmit PDO mapping 1/Statusword @bit 8
//     Drive/Inputs/In/nState4 @bit 1 <-> WcState/InputToggle
//     Drive/Inputs/In/nState4 <-> WcState/WcState
//     Drive/Inputs/In/nState5 <-> Transmit PDO mapping 1/Modes of operation display
//     Drive/Outputs/Out/nCtrl1 <-> Receive PDO mapping 1/Controlword
//     Drive/Outputs/Out/nCtrl2 <-> Receive PDO mapping 1/Controlword @bit 8
//     Drive/Outputs/Out/nCtrl5 <-> Receive PDO mapping 1/Modes of operation
//     Drive/Outputs/Out/nDataOut1 <-> Receive PDO mapping 1/Target position
//     Enc/Inputs/In/nDataIn1 <-> Transmit PDO mapping 1/Position actual value
//     Enc/Inputs/In/nDataIn3 <-> Transmit PDO mapping 1/Touch probe pos1 pos value
//     Enc/Inputs/In/nDcInputTime <-> InfoData/DcInputShift
//     Enc/Inputs/In/nState4 @bit 1 <-> WcState/InputToggle
//     Enc/Inputs/In/nState4 <-> WcState/WcState
//     Enc/Inputs/In/nState5 <-> Transmit PDO mapping 1/Touch probe status
//     Enc/Inputs/In/nState6 <-> Transmit PDO mapping 1/Touch probe status @bit 8
//     Enc/Outputs/Out/nCtrl5 <-> Receive PDO mapping 1/Touch probe function
//     Enc/Outputs/Out/nCtrl6 <-> Receive PDO mapping 1/Touch probe function @bit 8
//   NC-Task 1 SAF/Axes/Axis 5|OutRobot_X <-> Device 5 (EtherCAT)/Drive 42 (MADLT15BF)
//     Drive/Inputs/In/nDataIn1 <-> Transmit PDO mapping 1/Following error actual value
//     Drive/Inputs/In/nDcOutputTime <-> InfoData/DcOutputShift
//     Drive/Inputs/In/nState1 <-> Transmit PDO mapping 1/Statusword
//     Drive/Inputs/In/nState2 <-> Transmit PDO mapping 1/Statusword @bit 8
//     Drive/Inputs/In/nState4 @bit 1 <-> WcState/InputToggle
//     Drive/Inputs/In/nState4 <-> WcState/WcState
//     Drive/Inputs/In/nState5 <-> Transmit PDO mapping 1/Modes of operation display
//     Drive/Outputs/Out/nCtrl1 <-> Receive PDO mapping 1/Controlword
//     Drive/Outputs/Out/nCtrl2 <-> Receive PDO mapping 1/Controlword @bit 8
//     Drive/Outputs/Out/nCtrl5 <-> Receive PDO mapping 1/Modes of operation
//     Drive/Outputs/Out/nDataOut1 <-> Receive PDO mapping 1/Target position
//     Enc/Inputs/In/nDataIn1 <-> Transmit PDO mapping 1/Position actual value
//     Enc/Inputs/In/nDataIn3 <-> Transmit PDO mapping 1/Touch probe pos1 pos value
//     Enc/Inputs/In/nDcInputTime <-> InfoData/DcInputShift
//     Enc/Inputs/In/nState4 @bit 1 <-> WcState/InputToggle
//     Enc/Inputs/In/nState4 <-> WcState/WcState
//     Enc/Inputs/In/nState5 <-> Transmit PDO mapping 1/Touch probe status
//     Enc/Inputs/In/nState6 <-> Transmit PDO mapping 1/Touch probe status @bit 8
//     Enc/Outputs/Out/nCtrl5 <-> Receive PDO mapping 1/Touch probe function
//     Enc/Outputs/Out/nCtrl6 <-> Receive PDO mapping 1/Touch probe function @bit 8
//   NC-Task 1 SAF/Axes/Axis 6|OutRobot_Y <-> Device 5 (EtherCAT)/Drive 43 (MBDLT25BF)
//     Drive/Inputs/In/nDataIn1 <-> Transmit PDO mapping 1/Following error actual value
//     Drive/Inputs/In/nDcOutputTime <-> InfoData/DcOutputShift
//     Drive/Inputs/In/nState1 <-> Transmit PDO mapping 1/Statusword
//     Drive/Inputs/In/nState2 <-> Transmit PDO mapping 1/Statusword @bit 8
//     Drive/Inputs/In/nState4 @bit 1 <-> WcState/InputToggle
//     Drive/Inputs/In/nState4 <-> WcState/WcState
//     Drive/Inputs/In/nState5 <-> Transmit PDO mapping 1/Modes of operation display
//     Drive/Outputs/Out/nCtrl1 <-> Receive PDO mapping 1/Controlword
//     Drive/Outputs/Out/nCtrl2 <-> Receive PDO mapping 1/Controlword @bit 8
//     Drive/Outputs/Out/nCtrl5 <-> Receive PDO mapping 1/Modes of operation
//     Drive/Outputs/Out/nDataOut1 <-> Receive PDO mapping 1/Target position
//     Enc/Inputs/In/nDataIn1 <-> Transmit PDO mapping 1/Position actual value
//     Enc/Inputs/In/nDataIn3 <-> Transmit PDO mapping 1/Touch probe pos1 pos value
//     Enc/Inputs/In/nDcInputTime <-> InfoData/DcInputShift
//     Enc/Inputs/In/nState4 @bit 1 <-> WcState/InputToggle
//     Enc/Inputs/In/nState4 <-> WcState/WcState
//     Enc/Inputs/In/nState5 <-> Transmit PDO mapping 1/Touch probe status
//     Enc/Inputs/In/nState6 <-> Transmit PDO mapping 1/Touch probe status @bit 8
//     Enc/Outputs/Out/nCtrl5 <-> Receive PDO mapping 1/Touch probe function
//     Enc/Outputs/Out/nCtrl6 <-> Receive PDO mapping 1/Touch probe function @bit 8
//   NC-Task 1 SAF/Axes/Axis 7|RackMotor <-> Device 1 (EtherCAT) Storage/Term 1 (EK1200)/Term 18 (EL7342)
//     Drive/Inputs/In/nState1 @bit 3 <-> DCM Status Channel 1/Status/Error
//     Drive/Inputs/In/nState1 @bit 5 <-> DCM Status Channel 1/Status/Moving negative
//     Drive/Inputs/In/nState1 @bit 4 <-> DCM Status Channel 1/Status/Moving positive
//     Drive/Inputs/In/nState1 @bit 1 <-> DCM Status Channel 1/Status/Ready
//     Drive/Inputs/In/nState1 <-> DCM Status Channel 1/Status/Ready to enable
//     Drive/Inputs/In/nState1 @bit 6 <-> DCM Status Channel 1/Status/Torque reduced
//     Drive/Inputs/In/nState1 @bit 2 <-> DCM Status Channel 1/Status/Warning
//     Drive/Inputs/In/nState2 @bit 3 <-> DCM Status Channel 1/Status/Digital input 1
//     Drive/Inputs/In/nState2 @bit 4 <-> DCM Status Channel 1/Status/Digital input 2
//     Drive/Inputs/In/nState2 @bit 5 <-> DCM Status Channel 1/Status/Sync error
//     Drive/Inputs/In/nState2 @bit 7 <-> DCM Status Channel 1/Status/TxPDO Toggle
//     Drive/Inputs/In/nState4 @bit 1 <-> WcState/InputToggle
//     Drive/Inputs/In/nState4 <-> WcState/WcState
//     Drive/Outputs/Out/nCtrl1 <-> DCM Control Channel 1/Control/Enable
//     Drive/Outputs/Out/nCtrl1 @bit 2 <-> DCM Control Channel 1/Control/Reduce torque
//     Drive/Outputs/Out/nCtrl1 @bit 1 <-> DCM Control Channel 1/Control/Reset
//     Drive/Outputs/Out/nCtrl1 @bit 3 <-> DCM Control Channel 1/Control/Threshold active
//     Drive/Outputs/Out/nDataOut2[0] <-> DCM Velocity Channel 1/Velocity
//     Enc/Inputs/In/nDataIn1 <-> ENC Status Channel 1/Counter value
//     Enc/Inputs/In/nDataIn2 <-> ENC Status Channel 1/Latch value
//     Enc/Inputs/In/nState1 @bit 4 <-> ENC Status Channel 1/Status/Counter overflow
//     Enc/Inputs/In/nState1 @bit 3 <-> ENC Status Channel 1/Status/Counter underflow
//     Enc/Inputs/In/nState1 @bit 7 <-> ENC Status Channel 1/Status/Extrapolation stall
//     Enc/Inputs/In/nState1 @bit 1 <-> ENC Status Channel 1/Status/Latch extern valid
//     Enc/Inputs/In/nState1 @bit 2 <-> ENC Status Channel 1/Status/Set counter done
//     Enc/Inputs/In/nState2 @bit 4 <-> ENC Status Channel 1/Status/Status of extern latch
//     Enc/Inputs/In/nState2 <-> ENC Status Channel 1/Status/Status of input A
//     Enc/Inputs/In/nState2 @bit 1 <-> ENC Status Channel 1/Status/Status of input B
//     Enc/Inputs/In/nState2 @bit 5 <-> ENC Status Channel 1/Status/Sync error
//     Enc/Inputs/In/nState2 @bit 7 <-> ENC Status Channel 1/Status/TxPDO Toggle
//     Enc/Inputs/In/nState4 @bit 1 <-> WcState/InputToggle
//     Enc/Inputs/In/nState4 <-> WcState/WcState
//     Enc/Outputs/Out/nCtrl1 @bit 3 <-> ENC Control Channel 1/Control/Enable latch extern on negative edge
//     Enc/Outputs/Out/nCtrl1 @bit 1 <-> ENC Control Channel 1/Control/Enable latch extern on positive edge
//     Enc/Outputs/Out/nCtrl1 @bit 2 <-> ENC Control Channel 1/Control/Set counter
//     Enc/Outputs/Out/nDataOut1 <-> ENC Control Channel 1/Set counter value
//   DAS_CoreSys/DAS_CoreSys Instance <-> Device 1 (EtherCAT) Storage/Term 1 (EK1200)/Term 10 (EL2889)_01(Y4)
//     ModbusTask Outputs/GVL_Output.uniDO.stEbusDO.EL2889_01.DO1 <-> Channel 1/Output
//     ModbusTask Outputs/GVL_Output.uniDO.stEbusDO.EL2889_01.DO10 <-> Channel 10/Output
//     ModbusTask Outputs/GVL_Output.uniDO.stEbusDO.EL2889_01.DO11 <-> Channel 11/Output
//     ModbusTask Outputs/GVL_Output.uniDO.stEbusDO.EL2889_01.DO12 <-> Channel 12/Output
//     ModbusTask Outputs/GVL_Output.uniDO.stEbusDO.EL2889_01.DO13 <-> Channel 13/Output
//     ModbusTask Outputs/GVL_Output.uniDO.stEbusDO.EL2889_01.DO14 <-> Channel 14/Output
//     ModbusTask Outputs/GVL_Output.uniDO.stEbusDO.EL2889_01.DO15 <-> Channel 15/Output
//     ModbusTask Outputs/GVL_Output.uniDO.stEbusDO.EL2889_01.DO16 <-> Channel 16/Output
//     ModbusTask Outputs/GVL_Output.uniDO.stEbusDO.EL2889_01.DO2 <-> Channel 2/Output
//     ModbusTask Outputs/GVL_Output.uniDO.stEbusDO.EL2889_01.DO3 <-> Channel 3/Output
//     ModbusTask Outputs/GVL_Output.uniDO.stEbusDO.EL2889_01.DO4 <-> Channel 4/Output
//     ModbusTask Outputs/GVL_Output.uniDO.stEbusDO.EL2889_01.DO5 <-> Channel 5/Output
//     ModbusTask Outputs/GVL_Output.uniDO.stEbusDO.EL2889_01.DO6 <-> Channel 6/Output
//     ModbusTask Outputs/GVL_Output.uniDO.stEbusDO.EL2889_01.DO7 <-> Channel 7/Output
//     ModbusTask Outputs/GVL_Output.uniDO.stEbusDO.EL2889_01.DO8 <-> Channel 8/Output
//     ModbusTask Outputs/GVL_Output.uniDO.stEbusDO.EL2889_01.DO9 <-> Channel 9/Output
//   DAS_CoreSys/DAS_CoreSys Instance <-> Device 1 (EtherCAT) Storage/Term 1 (EK1200)/Term 11 (EL2889)_02(Y5)
//     ModbusTask Outputs/GVL_Output.uniDO.stEbusDO.EL2889_02.DO1 <-> Channel 1/Output
//     ModbusTask Outputs/GVL_Output.uniDO.stEbusDO.EL2889_02.DO10 <-> Channel 10/Output
//     ModbusTask Outputs/GVL_Output.uniDO.stEbusDO.EL2889_02.DO11 <-> Channel 11/Output
//     ModbusTask Outputs/GVL_Output.uniDO.stEbusDO.EL2889_02.DO12 <-> Channel 12/Output
//     ModbusTask Outputs/GVL_Output.uniDO.stEbusDO.EL2889_02.DO13 <-> Channel 13/Output
//     ModbusTask Outputs/GVL_Output.uniDO.stEbusDO.EL2889_02.DO14 <-> Channel 14/Output
//     ModbusTask Outputs/GVL_Output.uniDO.stEbusDO.EL2889_02.DO15 <-> Channel 15/Output
//     ModbusTask Outputs/GVL_Output.uniDO.stEbusDO.EL2889_02.DO16 <-> Channel 16/Output
//     ModbusTask Outputs/GVL_Output.uniDO.stEbusDO.EL2889_02.DO2 <-> Channel 2/Output
//     ModbusTask Outputs/GVL_Output.uniDO.stEbusDO.EL2889_02.DO3 <-> Channel 3/Output
//     ModbusTask Outputs/GVL_Output.uniDO.stEbusDO.EL2889_02.DO4 <-> Channel 4/Output
//     ModbusTask Outputs/GVL_Output.uniDO.stEbusDO.EL2889_02.DO5 <-> Channel 5/Output
//     ModbusTask Outputs/GVL_Output.uniDO.stEbusDO.EL2889_02.DO6 <-> Channel 6/Output
//     ModbusTask Outputs/GVL_Output.uniDO.stEbusDO.EL2889_02.DO7 <-> Channel 7/Output
//     ModbusTask Outputs/GVL_Output.uniDO.stEbusDO.EL2889_02.DO8 <-> Channel 8/Output
//     ModbusTask Outputs/GVL_Output.uniDO.stEbusDO.EL2889_02.DO9 <-> Channel 9/Output
//   DAS_CoreSys/DAS_CoreSys Instance <-> Device 1 (EtherCAT) Storage/Term 1 (EK1200)/Term 12 (EL2889)_03(Y6)
//     ModbusTask Outputs/GVL_Output.uniDO.stEbusDO.EL2889_03.DO1 <-> Channel 1/Output
//     ModbusTask Outputs/GVL_Output.uniDO.stEbusDO.EL2889_03.DO10 <-> Channel 10/Output
//     ModbusTask Outputs/GVL_Output.uniDO.stEbusDO.EL2889_03.DO11 <-> Channel 11/Output
//     ModbusTask Outputs/GVL_Output.uniDO.stEbusDO.EL2889_03.DO12 <-> Channel 12/Output
//     ModbusTask Outputs/GVL_Output.uniDO.stEbusDO.EL2889_03.DO13 <-> Channel 13/Output
//     ModbusTask Outputs/GVL_Output.uniDO.stEbusDO.EL2889_03.DO14 <-> Channel 14/Output
//     ModbusTask Outputs/GVL_Output.uniDO.stEbusDO.EL2889_03.DO15 <-> Channel 15/Output
//     ModbusTask Outputs/GVL_Output.uniDO.stEbusDO.EL2889_03.DO16 <-> Channel 16/Output
//     ModbusTask Outputs/GVL_Output.uniDO.stEbusDO.EL2889_03.DO2 <-> Channel 2/Output
//     ModbusTask Outputs/GVL_Output.uniDO.stEbusDO.EL2889_03.DO3 <-> Channel 3/Output
//     ModbusTask Outputs/GVL_Output.uniDO.stEbusDO.EL2889_03.DO4 <-> Channel 4/Output
//     ModbusTask Outputs/GVL_Output.uniDO.stEbusDO.EL2889_03.DO5 <-> Channel 5/Output
//     ModbusTask Outputs/GVL_Output.uniDO.stEbusDO.EL2889_03.DO6 <-> Channel 6/Output
//     ModbusTask Outputs/GVL_Output.uniDO.stEbusDO.EL2889_03.DO7 <-> Channel 7/Output
//     ModbusTask Outputs/GVL_Output.uniDO.stEbusDO.EL2889_03.DO8 <-> Channel 8/Output
//     ModbusTask Outputs/GVL_Output.uniDO.stEbusDO.EL2889_03.DO9 <-> Channel 9/Output
//   DAS_CoreSys/DAS_CoreSys Instance <-> Device 1 (EtherCAT) Storage/Term 1 (EK1200)/Term 13 (EL2889)_04(Y7)
//     ModbusTask Outputs/GVL_Output.uniDO.stEbusDO.EL2889_04.DO1 <-> Channel 1/Output
//     ModbusTask Outputs/GVL_Output.uniDO.stEbusDO.EL2889_04.DO10 <-> Channel 10/Output
//     ModbusTask Outputs/GVL_Output.uniDO.stEbusDO.EL2889_04.DO11 <-> Channel 11/Output
//     ModbusTask Outputs/GVL_Output.uniDO.stEbusDO.EL2889_04.DO12 <-> Channel 12/Output
//     ModbusTask Outputs/GVL_Output.uniDO.stEbusDO.EL2889_04.DO13 <-> Channel 13/Output
//     ModbusTask Outputs/GVL_Output.uniDO.stEbusDO.EL2889_04.DO14 <-> Channel 14/Output
//     ModbusTask Outputs/GVL_Output.uniDO.stEbusDO.EL2889_04.DO15 <-> Channel 15/Output
//     ModbusTask Outputs/GVL_Output.uniDO.stEbusDO.EL2889_04.DO16 <-> Channel 16/Output
//     ModbusTask Outputs/GVL_Output.uniDO.stEbusDO.EL2889_04.DO2 <-> Channel 2/Output
//     ModbusTask Outputs/GVL_Output.uniDO.stEbusDO.EL2889_04.DO3 <-> Channel 3/Output
//     ModbusTask Outputs/GVL_Output.uniDO.stEbusDO.EL2889_04.DO4 <-> Channel 4/Output
//     ModbusTask Outputs/GVL_Output.uniDO.stEbusDO.EL2889_04.DO5 <-> Channel 5/Output
//     ModbusTask Outputs/GVL_Output.uniDO.stEbusDO.EL2889_04.DO6 <-> Channel 6/Output
//     ModbusTask Outputs/GVL_Output.uniDO.stEbusDO.EL2889_04.DO7 <-> Channel 7/Output
//     ModbusTask Outputs/GVL_Output.uniDO.stEbusDO.EL2889_04.DO8 <-> Channel 8/Output
//     ModbusTask Outputs/GVL_Output.uniDO.stEbusDO.EL2889_04.DO9 <-> Channel 9/Output
//   DAS_CoreSys/DAS_CoreSys Instance <-> Device 1 (EtherCAT) Storage/Term 1 (EK1200)/Term 14 (EL2889)_05(Y8)
//     ModbusTask Outputs/GVL_Output.uniDO.stEbusDO.EL2889_05.DO1 <-> Channel 1/Output
//     ModbusTask Outputs/GVL_Output.uniDO.stEbusDO.EL2889_05.DO10 <-> Channel 10/Output
//     ModbusTask Outputs/GVL_Output.uniDO.stEbusDO.EL2889_05.DO11 <-> Channel 11/Output
//     ModbusTask Outputs/GVL_Output.uniDO.stEbusDO.EL2889_05.DO12 <-> Channel 12/Output
//     ModbusTask Outputs/GVL_Output.uniDO.stEbusDO.EL2889_05.DO13 <-> Channel 13/Output
//     ModbusTask Outputs/GVL_Output.uniDO.stEbusDO.EL2889_05.DO14 <-> Channel 14/Output
//     ModbusTask Outputs/GVL_Output.uniDO.stEbusDO.EL2889_05.DO15 <-> Channel 15/Output
//     ModbusTask Outputs/GVL_Output.uniDO.stEbusDO.EL2889_05.DO16 <-> Channel 16/Output
//     ModbusTask Outputs/GVL_Output.uniDO.stEbusDO.EL2889_05.DO2 <-> Channel 2/Output
//     ModbusTask Outputs/GVL_Output.uniDO.stEbusDO.EL2889_05.DO3 <-> Channel 3/Output
//     ModbusTask Outputs/GVL_Output.uniDO.stEbusDO.EL2889_05.DO4 <-> Channel 4/Output
//     ModbusTask Outputs/GVL_Output.uniDO.stEbusDO.EL2889_05.DO5 <-> Channel 5/Output
//     ModbusTask Outputs/GVL_Output.uniDO.stEbusDO.EL2889_05.DO6 <-> Channel 6/Output
//     ModbusTask Outputs/GVL_Output.uniDO.stEbusDO.EL2889_05.DO7 <-> Channel 7/Output
//     ModbusTask Outputs/GVL_Output.uniDO.stEbusDO.EL2889_05.DO8 <-> Channel 8/Output
//     ModbusTask Outputs/GVL_Output.uniDO.stEbusDO.EL2889_05.DO9 <-> Channel 9/Output
//   DAS_CoreSys/DAS_CoreSys Instance <-> Device 1 (EtherCAT) Storage/Term 1 (EK1200)/Term 15 (EL2889)_06(Y10)
//     ModbusTask Outputs/GVL_Output.uniDO.stEbusDO.EL2889_06.DO1 <-> Channel 1/Output
//     ModbusTask Outputs/GVL_Output.uniDO.stEbusDO.EL2889_06.DO10 <-> Channel 10/Output
//     ModbusTask Outputs/GVL_Output.uniDO.stEbusDO.EL2889_06.DO11 <-> Channel 11/Output
//     ModbusTask Outputs/GVL_Output.uniDO.stEbusDO.EL2889_06.DO12 <-> Channel 12/Output
//     ModbusTask Outputs/GVL_Output.uniDO.stEbusDO.EL2889_06.DO13 <-> Channel 13/Output
//     ModbusTask Outputs/GVL_Output.uniDO.stEbusDO.EL2889_06.DO14 <-> Channel 14/Output
//     ModbusTask Outputs/GVL_Output.uniDO.stEbusDO.EL2889_06.DO15 <-> Channel 15/Output
//     ModbusTask Outputs/GVL_Output.uniDO.stEbusDO.EL2889_06.DO16 <-> Channel 16/Output
//     ModbusTask Outputs/GVL_Output.uniDO.stEbusDO.EL2889_06.DO2 <-> Channel 2/Output
//     ModbusTask Outputs/GVL_Output.uniDO.stEbusDO.EL2889_06.DO3 <-> Channel 3/Output
//     ModbusTask Outputs/GVL_Output.uniDO.stEbusDO.EL2889_06.DO4 <-> Channel 4/Output
//     ModbusTask Outputs/GVL_Output.uniDO.stEbusDO.EL2889_06.DO5 <-> Channel 5/Output
//     ModbusTask Outputs/GVL_Output.uniDO.stEbusDO.EL2889_06.DO6 <-> Channel 6/Output
//     ModbusTask Outputs/GVL_Output.uniDO.stEbusDO.EL2889_06.DO7 <-> Channel 7/Output
//     ModbusTask Outputs/GVL_Output.uniDO.stEbusDO.EL2889_06.DO8 <-> Channel 8/Output
//     ModbusTask Outputs/GVL_Output.uniDO.stEbusDO.EL2889_06.DO9 <-> Channel 9/Output
//   DAS_CoreSys/DAS_CoreSys Instance <-> Device 1 (EtherCAT) Storage/Term 1 (EK1200)/Term 17 (EL2889)_07(Y11)
//     ModbusTask Outputs/GVL_Output.uniDO.stEbusDO.EL2889_07.DO1 <-> Channel 1/Output
//     ModbusTask Outputs/GVL_Output.uniDO.stEbusDO.EL2889_07.DO10 <-> Channel 10/Output
//     ModbusTask Outputs/GVL_Output.uniDO.stEbusDO.EL2889_07.DO11 <-> Channel 11/Output
//     ModbusTask Outputs/GVL_Output.uniDO.stEbusDO.EL2889_07.DO12 <-> Channel 12/Output
//     ModbusTask Outputs/GVL_Output.uniDO.stEbusDO.EL2889_07.DO13 <-> Channel 13/Output
//     ModbusTask Outputs/GVL_Output.uniDO.stEbusDO.EL2889_07.DO14 <-> Channel 14/Output
//     ModbusTask Outputs/GVL_Output.uniDO.stEbusDO.EL2889_07.DO15 <-> Channel 15/Output
//     ModbusTask Outputs/GVL_Output.uniDO.stEbusDO.EL2889_07.DO16 <-> Channel 16/Output
//     ModbusTask Outputs/GVL_Output.uniDO.stEbusDO.EL2889_07.DO2 <-> Channel 2/Output
//     ModbusTask Outputs/GVL_Output.uniDO.stEbusDO.EL2889_07.DO3 <-> Channel 3/Output
//     ModbusTask Outputs/GVL_Output.uniDO.stEbusDO.EL2889_07.DO4 <-> Channel 4/Output
//     ModbusTask Outputs/GVL_Output.uniDO.stEbusDO.EL2889_07.DO5 <-> Channel 5/Output
//     ModbusTask Outputs/GVL_Output.uniDO.stEbusDO.EL2889_07.DO6 <-> Channel 6/Output
//     ModbusTask Outputs/GVL_Output.uniDO.stEbusDO.EL2889_07.DO7 <-> Channel 7/Output
//     ModbusTask Outputs/GVL_Output.uniDO.stEbusDO.EL2889_07.DO8 <-> Channel 8/Output
//     ModbusTask Outputs/GVL_Output.uniDO.stEbusDO.EL2889_07.DO9 <-> Channel 9/Output
//   DAS_CoreSys/DAS_CoreSys Instance <-> Device 1 (EtherCAT) Storage/Term 1 (EK1200)/Term 2 (EL6021)
//     ModbusTask Inputs/MAIN2_RS485.RS485_V2[4].ModbusRtuMasterV2_KL6x22B.InData/D <-> COM TxPDO-Map Inputs/Data In 0
//     ModbusTask Inputs/MAIN2_RS485.RS485_V2[4].ModbusRtuMasterV2_KL6x22B.InData/D @bit {8..168 step 8} <-> COM TxPDO-Map Inputs/Data In {1..21}  (21 links)
//     ModbusTask Inputs/MAIN2_RS485.RS485_V2[4].ModbusRtuMasterV2_KL6x22B.InData/Status <-> COM TxPDO-Map Inputs/Status
//     ModbusTask Outputs/MAIN2_RS485.RS485_V2[4].ModbusRtuMasterV2_KL6x22B.OutData/Ctrl <-> COM RxPDO-Map Outputs/Ctrl
//     ModbusTask Outputs/MAIN2_RS485.RS485_V2[4].ModbusRtuMasterV2_KL6x22B.OutData/D <-> COM RxPDO-Map Outputs/Data Out 0
//     ModbusTask Outputs/MAIN2_RS485.RS485_V2[4].ModbusRtuMasterV2_KL6x22B.OutData/D @bit {8..168 step 8} <-> COM RxPDO-Map Outputs/Data Out {1..21}  (21 links)
//   DAS_CoreSys/DAS_CoreSys Instance <-> Device 1 (EtherCAT) Storage/Term 1 (EK1200)/Term 3 (EL6021)
//     ModbusTask Inputs/MAIN2_RS485.RS485_V2[3].ModbusRtuMasterV2_KL6x22B.InData/D <-> COM TxPDO-Map Inputs/Data In 0
//     ModbusTask Inputs/MAIN2_RS485.RS485_V2[3].ModbusRtuMasterV2_KL6x22B.InData/D @bit {8..168 step 8} <-> COM TxPDO-Map Inputs/Data In {1..21}  (21 links)
//     ModbusTask Inputs/MAIN2_RS485.RS485_V2[3].ModbusRtuMasterV2_KL6x22B.InData/Status <-> COM TxPDO-Map Inputs/Status
//     ModbusTask Outputs/MAIN2_RS485.RS485_V2[3].ModbusRtuMasterV2_KL6x22B.OutData/Ctrl <-> COM RxPDO-Map Outputs/Ctrl
//     ModbusTask Outputs/MAIN2_RS485.RS485_V2[3].ModbusRtuMasterV2_KL6x22B.OutData/D <-> COM RxPDO-Map Outputs/Data Out 0
//     ModbusTask Outputs/MAIN2_RS485.RS485_V2[3].ModbusRtuMasterV2_KL6x22B.OutData/D @bit {8..168 step 8} <-> COM RxPDO-Map Outputs/Data Out {1..21}  (21 links)
//   DAS_CoreSys/DAS_CoreSys Instance <-> Device 1 (EtherCAT) Storage/Term 1 (EK1200)/Term 4 (EL6021)
//     ModbusTask Inputs/MAIN2_RS485.RS485_V2[2].ModbusRtuMasterV2_KL6x22B.InData/D <-> COM TxPDO-Map Inputs/Data In 0
//     ModbusTask Inputs/MAIN2_RS485.RS485_V2[2].ModbusRtuMasterV2_KL6x22B.InData/D @bit {8..168 step 8} <-> COM TxPDO-Map Inputs/Data In {1..21}  (21 links)
//     ModbusTask Inputs/MAIN2_RS485.RS485_V2[2].ModbusRtuMasterV2_KL6x22B.InData/Status <-> COM TxPDO-Map Inputs/Status
//     ModbusTask Outputs/MAIN2_RS485.RS485_V2[2].ModbusRtuMasterV2_KL6x22B.OutData/Ctrl <-> COM RxPDO-Map Outputs/Ctrl
//     ModbusTask Outputs/MAIN2_RS485.RS485_V2[2].ModbusRtuMasterV2_KL6x22B.OutData/D <-> COM RxPDO-Map Outputs/Data Out 0
//     ModbusTask Outputs/MAIN2_RS485.RS485_V2[2].ModbusRtuMasterV2_KL6x22B.OutData/D @bit {8..168 step 8} <-> COM RxPDO-Map Outputs/Data Out {1..21}  (21 links)
//   DAS_CoreSys/DAS_CoreSys Instance <-> Device 1 (EtherCAT) Storage/Term 1 (EK1200)/Term 5 (EL6021)
//     ModbusTask Inputs/MAIN2_RS485.RS485_V2[1].ModbusRtuMasterV2_KL6x22B.InData/D <-> COM TxPDO-Map Inputs/Data In 0
//     ModbusTask Inputs/MAIN2_RS485.RS485_V2[1].ModbusRtuMasterV2_KL6x22B.InData/D @bit {8..168 step 8} <-> COM TxPDO-Map Inputs/Data In {1..21}  (21 links)
//     ModbusTask Inputs/MAIN2_RS485.RS485_V2[1].ModbusRtuMasterV2_KL6x22B.InData/Status <-> COM TxPDO-Map Inputs/Status
//     ModbusTask Outputs/MAIN2_RS485.RS485_V2[1].ModbusRtuMasterV2_KL6x22B.OutData/Ctrl <-> COM RxPDO-Map Outputs/Ctrl
//     ModbusTask Outputs/MAIN2_RS485.RS485_V2[1].ModbusRtuMasterV2_KL6x22B.OutData/D <-> COM RxPDO-Map Outputs/Data Out 0
//     ModbusTask Outputs/MAIN2_RS485.RS485_V2[1].ModbusRtuMasterV2_KL6x22B.OutData/D @bit {8..168 step 8} <-> COM RxPDO-Map Outputs/Data Out {1..21}  (21 links)
//   DAS_CoreSys/DAS_CoreSys Instance <-> Device 1 (EtherCAT) Storage/Term 1 (EK1200)/Term 6 (EL1889)_01(X6)
//     ModbusTask Inputs/GVL_Input.uniDI.stEbusDI.EL1889_01.DI1 <-> Channel 1/Input
//     ModbusTask Inputs/GVL_Input.uniDI.stEbusDI.EL1889_01.DI10 <-> Channel 10/Input
//     ModbusTask Inputs/GVL_Input.uniDI.stEbusDI.EL1889_01.DI11 <-> Channel 11/Input
//     ModbusTask Inputs/GVL_Input.uniDI.stEbusDI.EL1889_01.DI12 <-> Channel 12/Input
//     ModbusTask Inputs/GVL_Input.uniDI.stEbusDI.EL1889_01.DI13 <-> Channel 13/Input
//     ModbusTask Inputs/GVL_Input.uniDI.stEbusDI.EL1889_01.DI14 <-> Channel 14/Input
//     ModbusTask Inputs/GVL_Input.uniDI.stEbusDI.EL1889_01.DI15 <-> Channel 15/Input
//     ModbusTask Inputs/GVL_Input.uniDI.stEbusDI.EL1889_01.DI16 <-> Channel 16/Input
//     ModbusTask Inputs/GVL_Input.uniDI.stEbusDI.EL1889_01.DI2 <-> Channel 2/Input
//     ModbusTask Inputs/GVL_Input.uniDI.stEbusDI.EL1889_01.DI3 <-> Channel 3/Input
//     ModbusTask Inputs/GVL_Input.uniDI.stEbusDI.EL1889_01.DI4 <-> Channel 4/Input
//     ModbusTask Inputs/GVL_Input.uniDI.stEbusDI.EL1889_01.DI5 <-> Channel 5/Input
//     ModbusTask Inputs/GVL_Input.uniDI.stEbusDI.EL1889_01.DI6 <-> Channel 6/Input
//     ModbusTask Inputs/GVL_Input.uniDI.stEbusDI.EL1889_01.DI7 <-> Channel 7/Input
//     ModbusTask Inputs/GVL_Input.uniDI.stEbusDI.EL1889_01.DI8 <-> Channel 8/Input
//     ModbusTask Inputs/GVL_Input.uniDI.stEbusDI.EL1889_01.DI9 <-> Channel 9/Input
//   DAS_CoreSys/DAS_CoreSys Instance <-> Device 1 (EtherCAT) Storage/Term 1 (EK1200)/Term 7 (EL1889)_02(X7)
//     ModbusTask Inputs/GVL_Input.uniDI.stEbusDI.EL1889_02.DI1 <-> Channel 1/Input
//     ModbusTask Inputs/GVL_Input.uniDI.stEbusDI.EL1889_02.DI10 <-> Channel 10/Input
//     ModbusTask Inputs/GVL_Input.uniDI.stEbusDI.EL1889_02.DI11 <-> Channel 11/Input
//     ModbusTask Inputs/GVL_Input.uniDI.stEbusDI.EL1889_02.DI12 <-> Channel 12/Input
//     ModbusTask Inputs/GVL_Input.uniDI.stEbusDI.EL1889_02.DI13 <-> Channel 13/Input
//     ModbusTask Inputs/GVL_Input.uniDI.stEbusDI.EL1889_02.DI14 <-> Channel 14/Input
//     ModbusTask Inputs/GVL_Input.uniDI.stEbusDI.EL1889_02.DI15 <-> Channel 15/Input
//     ModbusTask Inputs/GVL_Input.uniDI.stEbusDI.EL1889_02.DI16 <-> Channel 16/Input
//     ModbusTask Inputs/GVL_Input.uniDI.stEbusDI.EL1889_02.DI2 <-> Channel 2/Input
//     ModbusTask Inputs/GVL_Input.uniDI.stEbusDI.EL1889_02.DI3 <-> Channel 3/Input
//     ModbusTask Inputs/GVL_Input.uniDI.stEbusDI.EL1889_02.DI4 <-> Channel 4/Input
//     ModbusTask Inputs/GVL_Input.uniDI.stEbusDI.EL1889_02.DI5 <-> Channel 5/Input
//     ModbusTask Inputs/GVL_Input.uniDI.stEbusDI.EL1889_02.DI6 <-> Channel 6/Input
//     ModbusTask Inputs/GVL_Input.uniDI.stEbusDI.EL1889_02.DI7 <-> Channel 7/Input
//     ModbusTask Inputs/GVL_Input.uniDI.stEbusDI.EL1889_02.DI8 <-> Channel 8/Input
//     ModbusTask Inputs/GVL_Input.uniDI.stEbusDI.EL1889_02.DI9 <-> Channel 9/Input
//   DAS_CoreSys/DAS_CoreSys Instance <-> Device 1 (EtherCAT) Storage/Term 1 (EK1200)/Term 8 (EL1889)_03(X9)
//     ModbusTask Inputs/GVL_Input.uniDI.stEbusDI.EL1889_03.DI1 <-> Channel 1/Input
//     ModbusTask Inputs/GVL_Input.uniDI.stEbusDI.EL1889_03.DI10 <-> Channel 10/Input
//     ModbusTask Inputs/GVL_Input.uniDI.stEbusDI.EL1889_03.DI11 <-> Channel 11/Input
//     ModbusTask Inputs/GVL_Input.uniDI.stEbusDI.EL1889_03.DI12 <-> Channel 12/Input
//     ModbusTask Inputs/GVL_Input.uniDI.stEbusDI.EL1889_03.DI13 <-> Channel 13/Input
//     ModbusTask Inputs/GVL_Input.uniDI.stEbusDI.EL1889_03.DI14 <-> Channel 14/Input
//     ModbusTask Inputs/GVL_Input.uniDI.stEbusDI.EL1889_03.DI15 <-> Channel 15/Input
//     ModbusTask Inputs/GVL_Input.uniDI.stEbusDI.EL1889_03.DI16 <-> Channel 16/Input
//     ModbusTask Inputs/GVL_Input.uniDI.stEbusDI.EL1889_03.DI2 <-> Channel 2/Input
//     ModbusTask Inputs/GVL_Input.uniDI.stEbusDI.EL1889_03.DI3 <-> Channel 3/Input
//     ModbusTask Inputs/GVL_Input.uniDI.stEbusDI.EL1889_03.DI4 <-> Channel 4/Input
//     ModbusTask Inputs/GVL_Input.uniDI.stEbusDI.EL1889_03.DI5 <-> Channel 5/Input
//     ModbusTask Inputs/GVL_Input.uniDI.stEbusDI.EL1889_03.DI6 <-> Channel 6/Input
//     ModbusTask Inputs/GVL_Input.uniDI.stEbusDI.EL1889_03.DI7 <-> Channel 7/Input
//     ModbusTask Inputs/GVL_Input.uniDI.stEbusDI.EL1889_03.DI8 <-> Channel 8/Input
//     ModbusTask Inputs/GVL_Input.uniDI.stEbusDI.EL1889_03.DI9 <-> Channel 9/Input
//   DAS_CoreSys/DAS_CoreSys Instance <-> Device 1 (EtherCAT) Storage/Term 1 (EK1200)/Term 9 (EL1889)_04(X10)
//     ModbusTask Inputs/GVL_Input.uniDI.stEbusDI.EL1889_04.DI1 <-> Channel 1/Input
//     ModbusTask Inputs/GVL_Input.uniDI.stEbusDI.EL1889_04.DI10 <-> Channel 10/Input
//     ModbusTask Inputs/GVL_Input.uniDI.stEbusDI.EL1889_04.DI11 <-> Channel 11/Input
//     ModbusTask Inputs/GVL_Input.uniDI.stEbusDI.EL1889_04.DI12 <-> Channel 12/Input
//     ModbusTask Inputs/GVL_Input.uniDI.stEbusDI.EL1889_04.DI13 <-> Channel 13/Input
//     ModbusTask Inputs/GVL_Input.uniDI.stEbusDI.EL1889_04.DI14 <-> Channel 14/Input
//     ModbusTask Inputs/GVL_Input.uniDI.stEbusDI.EL1889_04.DI15 <-> Channel 15/Input
//     ModbusTask Inputs/GVL_Input.uniDI.stEbusDI.EL1889_04.DI16 <-> Channel 16/Input
//     ModbusTask Inputs/GVL_Input.uniDI.stEbusDI.EL1889_04.DI2 <-> Channel 2/Input
//     ModbusTask Inputs/GVL_Input.uniDI.stEbusDI.EL1889_04.DI3 <-> Channel 3/Input
//     ModbusTask Inputs/GVL_Input.uniDI.stEbusDI.EL1889_04.DI4 <-> Channel 4/Input
//     ModbusTask Inputs/GVL_Input.uniDI.stEbusDI.EL1889_04.DI5 <-> Channel 5/Input
//     ModbusTask Inputs/GVL_Input.uniDI.stEbusDI.EL1889_04.DI6 <-> Channel 6/Input
//     ModbusTask Inputs/GVL_Input.uniDI.stEbusDI.EL1889_04.DI7 <-> Channel 7/Input
//     ModbusTask Inputs/GVL_Input.uniDI.stEbusDI.EL1889_04.DI8 <-> Channel 8/Input
//     ModbusTask Inputs/GVL_Input.uniDI.stEbusDI.EL1889_04.DI9 <-> Channel 9/Input
//   DAS_CoreSys/DAS_CoreSys Instance <-> Device 4 (EtherCAT) Allocate/Term 22 (EK1100)/Term 23 (EL1889)_05(X0)
//     ModbusTask Inputs/GVL_Input.uniDI.stEbusDI.EL1889_05.DI1 <-> Channel 1/Input
//     ModbusTask Inputs/GVL_Input.uniDI.stEbusDI.EL1889_05.DI10 <-> Channel 10/Input
//     ModbusTask Inputs/GVL_Input.uniDI.stEbusDI.EL1889_05.DI11 <-> Channel 11/Input
//     ModbusTask Inputs/GVL_Input.uniDI.stEbusDI.EL1889_05.DI12 <-> Channel 12/Input
//     ModbusTask Inputs/GVL_Input.uniDI.stEbusDI.EL1889_05.DI13 <-> Channel 13/Input
//     ModbusTask Inputs/GVL_Input.uniDI.stEbusDI.EL1889_05.DI14 <-> Channel 14/Input
//     ModbusTask Inputs/GVL_Input.uniDI.stEbusDI.EL1889_05.DI15 <-> Channel 15/Input
//     ModbusTask Inputs/GVL_Input.uniDI.stEbusDI.EL1889_05.DI16 <-> Channel 16/Input
//     ModbusTask Inputs/GVL_Input.uniDI.stEbusDI.EL1889_05.DI2 <-> Channel 2/Input
//     ModbusTask Inputs/GVL_Input.uniDI.stEbusDI.EL1889_05.DI3 <-> Channel 3/Input
//     ModbusTask Inputs/GVL_Input.uniDI.stEbusDI.EL1889_05.DI4 <-> Channel 4/Input
//     ModbusTask Inputs/GVL_Input.uniDI.stEbusDI.EL1889_05.DI5 <-> Channel 5/Input
//     ModbusTask Inputs/GVL_Input.uniDI.stEbusDI.EL1889_05.DI6 <-> Channel 6/Input
//     ModbusTask Inputs/GVL_Input.uniDI.stEbusDI.EL1889_05.DI7 <-> Channel 7/Input
//     ModbusTask Inputs/GVL_Input.uniDI.stEbusDI.EL1889_05.DI8 <-> Channel 8/Input
//     ModbusTask Inputs/GVL_Input.uniDI.stEbusDI.EL1889_05.DI9 <-> Channel 9/Input
//   DAS_CoreSys/DAS_CoreSys Instance <-> Device 4 (EtherCAT) Allocate/Term 22 (EK1100)/Term 24 (EL1889)_06(X1)
//     ModbusTask Inputs/GVL_Input.uniDI.stEbusDI.EL1889_06.DI1 <-> Channel 1/Input
//     ModbusTask Inputs/GVL_Input.uniDI.stEbusDI.EL1889_06.DI10 <-> Channel 10/Input
//     ModbusTask Inputs/GVL_Input.uniDI.stEbusDI.EL1889_06.DI11 <-> Channel 11/Input
//     ModbusTask Inputs/GVL_Input.uniDI.stEbusDI.EL1889_06.DI12 <-> Channel 12/Input
//     ModbusTask Inputs/GVL_Input.uniDI.stEbusDI.EL1889_06.DI13 <-> Channel 13/Input
//     ModbusTask Inputs/GVL_Input.uniDI.stEbusDI.EL1889_06.DI14 <-> Channel 14/Input
//     ModbusTask Inputs/GVL_Input.uniDI.stEbusDI.EL1889_06.DI15 <-> Channel 15/Input
//     ModbusTask Inputs/GVL_Input.uniDI.stEbusDI.EL1889_06.DI16 <-> Channel 16/Input
//     ModbusTask Inputs/GVL_Input.uniDI.stEbusDI.EL1889_06.DI2 <-> Channel 2/Input
//     ModbusTask Inputs/GVL_Input.uniDI.stEbusDI.EL1889_06.DI3 <-> Channel 3/Input
//     ModbusTask Inputs/GVL_Input.uniDI.stEbusDI.EL1889_06.DI4 <-> Channel 4/Input
//     ModbusTask Inputs/GVL_Input.uniDI.stEbusDI.EL1889_06.DI5 <-> Channel 5/Input
//     ModbusTask Inputs/GVL_Input.uniDI.stEbusDI.EL1889_06.DI6 <-> Channel 6/Input
//     ModbusTask Inputs/GVL_Input.uniDI.stEbusDI.EL1889_06.DI7 <-> Channel 7/Input
//     ModbusTask Inputs/GVL_Input.uniDI.stEbusDI.EL1889_06.DI8 <-> Channel 8/Input
//     ModbusTask Inputs/GVL_Input.uniDI.stEbusDI.EL1889_06.DI9 <-> Channel 9/Input
//   DAS_CoreSys/DAS_CoreSys Instance <-> Device 4 (EtherCAT) Allocate/Term 22 (EK1100)/Term 25 (EL1889)_07(X2)
//     ModbusTask Inputs/GVL_Input.uniDI.stEbusDI.EL1889_07.DI1 <-> Channel 1/Input
//     ModbusTask Inputs/GVL_Input.uniDI.stEbusDI.EL1889_07.DI10 <-> Channel 10/Input
//     ModbusTask Inputs/GVL_Input.uniDI.stEbusDI.EL1889_07.DI11 <-> Channel 11/Input
//     ModbusTask Inputs/GVL_Input.uniDI.stEbusDI.EL1889_07.DI12 <-> Channel 12/Input
//     ModbusTask Inputs/GVL_Input.uniDI.stEbusDI.EL1889_07.DI13 <-> Channel 13/Input
//     ModbusTask Inputs/GVL_Input.uniDI.stEbusDI.EL1889_07.DI14 <-> Channel 14/Input
//     ModbusTask Inputs/GVL_Input.uniDI.stEbusDI.EL1889_07.DI15 <-> Channel 15/Input
//     ModbusTask Inputs/GVL_Input.uniDI.stEbusDI.EL1889_07.DI16 <-> Channel 16/Input
//     ModbusTask Inputs/GVL_Input.uniDI.stEbusDI.EL1889_07.DI2 <-> Channel 2/Input
//     ModbusTask Inputs/GVL_Input.uniDI.stEbusDI.EL1889_07.DI3 <-> Channel 3/Input
//     ModbusTask Inputs/GVL_Input.uniDI.stEbusDI.EL1889_07.DI4 <-> Channel 4/Input
//     ModbusTask Inputs/GVL_Input.uniDI.stEbusDI.EL1889_07.DI5 <-> Channel 5/Input
//     ModbusTask Inputs/GVL_Input.uniDI.stEbusDI.EL1889_07.DI6 <-> Channel 6/Input
//     ModbusTask Inputs/GVL_Input.uniDI.stEbusDI.EL1889_07.DI7 <-> Channel 7/Input
//     ModbusTask Inputs/GVL_Input.uniDI.stEbusDI.EL1889_07.DI8 <-> Channel 8/Input
//     ModbusTask Inputs/GVL_Input.uniDI.stEbusDI.EL1889_07.DI9 <-> Channel 9/Input
//   DAS_CoreSys/DAS_CoreSys Instance <-> Device 4 (EtherCAT) Allocate/Term 22 (EK1100)/Term 26 (EL1889)_08(X3)
//     ModbusTask Inputs/GVL_Input.uniDI.stEbusDI.EL1889_08.DI1 <-> Channel 1/Input
//     ModbusTask Inputs/GVL_Input.uniDI.stEbusDI.EL1889_08.DI10 <-> Channel 10/Input
//     ModbusTask Inputs/GVL_Input.uniDI.stEbusDI.EL1889_08.DI11 <-> Channel 11/Input
//     ModbusTask Inputs/GVL_Input.uniDI.stEbusDI.EL1889_08.DI12 <-> Channel 12/Input
//     ModbusTask Inputs/GVL_Input.uniDI.stEbusDI.EL1889_08.DI13 <-> Channel 13/Input
//     ModbusTask Inputs/GVL_Input.uniDI.stEbusDI.EL1889_08.DI14 <-> Channel 14/Input
//     ModbusTask Inputs/GVL_Input.uniDI.stEbusDI.EL1889_08.DI15 <-> Channel 15/Input
//     ModbusTask Inputs/GVL_Input.uniDI.stEbusDI.EL1889_08.DI16 <-> Channel 16/Input
//     ModbusTask Inputs/GVL_Input.uniDI.stEbusDI.EL1889_08.DI2 <-> Channel 2/Input
//     ModbusTask Inputs/GVL_Input.uniDI.stEbusDI.EL1889_08.DI3 <-> Channel 3/Input
//     ModbusTask Inputs/GVL_Input.uniDI.stEbusDI.EL1889_08.DI4 <-> Channel 4/Input
//     ModbusTask Inputs/GVL_Input.uniDI.stEbusDI.EL1889_08.DI5 <-> Channel 5/Input
//     ModbusTask Inputs/GVL_Input.uniDI.stEbusDI.EL1889_08.DI6 <-> Channel 6/Input
//     ModbusTask Inputs/GVL_Input.uniDI.stEbusDI.EL1889_08.DI7 <-> Channel 7/Input
//     ModbusTask Inputs/GVL_Input.uniDI.stEbusDI.EL1889_08.DI8 <-> Channel 8/Input
//     ModbusTask Inputs/GVL_Input.uniDI.stEbusDI.EL1889_08.DI9 <-> Channel 9/Input
//   DAS_CoreSys/DAS_CoreSys Instance <-> Device 4 (EtherCAT) Allocate/Term 22 (EK1100)/Term 27 (EL1889)_09(X8)
//     ModbusTask Inputs/GVL_Input.uniDI.stEbusDI.EL1889_09.DI1 <-> Channel 1/Input
//     ModbusTask Inputs/GVL_Input.uniDI.stEbusDI.EL1889_09.DI10 <-> Channel 10/Input
//     ModbusTask Inputs/GVL_Input.uniDI.stEbusDI.EL1889_09.DI11 <-> Channel 11/Input
//     ModbusTask Inputs/GVL_Input.uniDI.stEbusDI.EL1889_09.DI12 <-> Channel 12/Input
//     ModbusTask Inputs/GVL_Input.uniDI.stEbusDI.EL1889_09.DI13 <-> Channel 13/Input
//     ModbusTask Inputs/GVL_Input.uniDI.stEbusDI.EL1889_09.DI14 <-> Channel 14/Input
//     ModbusTask Inputs/GVL_Input.uniDI.stEbusDI.EL1889_09.DI15 <-> Channel 15/Input
//     ModbusTask Inputs/GVL_Input.uniDI.stEbusDI.EL1889_09.DI16 <-> Channel 16/Input
//     ModbusTask Inputs/GVL_Input.uniDI.stEbusDI.EL1889_09.DI2 <-> Channel 2/Input
//     ModbusTask Inputs/GVL_Input.uniDI.stEbusDI.EL1889_09.DI3 <-> Channel 3/Input
//     ModbusTask Inputs/GVL_Input.uniDI.stEbusDI.EL1889_09.DI4 <-> Channel 4/Input
//     ModbusTask Inputs/GVL_Input.uniDI.stEbusDI.EL1889_09.DI5 <-> Channel 5/Input
//     ModbusTask Inputs/GVL_Input.uniDI.stEbusDI.EL1889_09.DI6 <-> Channel 6/Input
//     ModbusTask Inputs/GVL_Input.uniDI.stEbusDI.EL1889_09.DI7 <-> Channel 7/Input
//     ModbusTask Inputs/GVL_Input.uniDI.stEbusDI.EL1889_09.DI8 <-> Channel 8/Input
//     ModbusTask Inputs/GVL_Input.uniDI.stEbusDI.EL1889_09.DI9 <-> Channel 9/Input
//   DAS_CoreSys/DAS_CoreSys Instance <-> Device 4 (EtherCAT) Allocate/Term 22 (EK1100)/Term 28 (EL1889)_10(X11)
//     ModbusTask Inputs/GVL_Input.uniDI.stEbusDI.EL1889_10.DI{1..16} <-> Channel {1..16}/Input  (16 links)
//   DAS_CoreSys/DAS_CoreSys Instance <-> Device 4 (EtherCAT) Allocate/Term 22 (EK1100)/Term 29 (EL2889)_08(Y0)
//     ModbusTask Outputs/GVL_Output.uniDO.stEbusDO.EL2889_08.DO1 <-> Channel 1/Output
//     ModbusTask Outputs/GVL_Output.uniDO.stEbusDO.EL2889_08.DO10 <-> Channel 10/Output
//     ModbusTask Outputs/GVL_Output.uniDO.stEbusDO.EL2889_08.DO11 <-> Channel 11/Output
//     ModbusTask Outputs/GVL_Output.uniDO.stEbusDO.EL2889_08.DO12 <-> Channel 12/Output
//     ModbusTask Outputs/GVL_Output.uniDO.stEbusDO.EL2889_08.DO13 <-> Channel 13/Output
//     ModbusTask Outputs/GVL_Output.uniDO.stEbusDO.EL2889_08.DO14 <-> Channel 14/Output
//     ModbusTask Outputs/GVL_Output.uniDO.stEbusDO.EL2889_08.DO15 <-> Channel 15/Output
//     ModbusTask Outputs/GVL_Output.uniDO.stEbusDO.EL2889_08.DO16 <-> Channel 16/Output
//     ModbusTask Outputs/GVL_Output.uniDO.stEbusDO.EL2889_08.DO2 <-> Channel 2/Output
//     ModbusTask Outputs/GVL_Output.uniDO.stEbusDO.EL2889_08.DO3 <-> Channel 3/Output
//     ModbusTask Outputs/GVL_Output.uniDO.stEbusDO.EL2889_08.DO4 <-> Channel 4/Output
//     ModbusTask Outputs/GVL_Output.uniDO.stEbusDO.EL2889_08.DO5 <-> Channel 5/Output
//     ModbusTask Outputs/GVL_Output.uniDO.stEbusDO.EL2889_08.DO6 <-> Channel 6/Output
//     ModbusTask Outputs/GVL_Output.uniDO.stEbusDO.EL2889_08.DO7 <-> Channel 7/Output
//     ModbusTask Outputs/GVL_Output.uniDO.stEbusDO.EL2889_08.DO8 <-> Channel 8/Output
//     ModbusTask Outputs/GVL_Output.uniDO.stEbusDO.EL2889_08.DO9 <-> Channel 9/Output
//   DAS_CoreSys/DAS_CoreSys Instance <-> Device 4 (EtherCAT) Allocate/Term 22 (EK1100)/Term 30 (EL2889)_09(Y1)
//     ModbusTask Outputs/GVL_Output.uniDO.stEbusDO.EL2889_09.DO1 <-> Channel 1/Output
//     ModbusTask Outputs/GVL_Output.uniDO.stEbusDO.EL2889_09.DO10 <-> Channel 10/Output
//     ModbusTask Outputs/GVL_Output.uniDO.stEbusDO.EL2889_09.DO11 <-> Channel 11/Output
//     ModbusTask Outputs/GVL_Output.uniDO.stEbusDO.EL2889_09.DO12 <-> Channel 12/Output
//     ModbusTask Outputs/GVL_Output.uniDO.stEbusDO.EL2889_09.DO13 <-> Channel 13/Output
//     ModbusTask Outputs/GVL_Output.uniDO.stEbusDO.EL2889_09.DO14 <-> Channel 14/Output
//     ModbusTask Outputs/GVL_Output.uniDO.stEbusDO.EL2889_09.DO15 <-> Channel 15/Output
//     ModbusTask Outputs/GVL_Output.uniDO.stEbusDO.EL2889_09.DO16 <-> Channel 16/Output
//     ModbusTask Outputs/GVL_Output.uniDO.stEbusDO.EL2889_09.DO2 <-> Channel 2/Output
//     ModbusTask Outputs/GVL_Output.uniDO.stEbusDO.EL2889_09.DO3 <-> Channel 3/Output
//     ModbusTask Outputs/GVL_Output.uniDO.stEbusDO.EL2889_09.DO4 <-> Channel 4/Output
//     ModbusTask Outputs/GVL_Output.uniDO.stEbusDO.EL2889_09.DO5 <-> Channel 5/Output
//     ModbusTask Outputs/GVL_Output.uniDO.stEbusDO.EL2889_09.DO6 <-> Channel 6/Output
//     ModbusTask Outputs/GVL_Output.uniDO.stEbusDO.EL2889_09.DO7 <-> Channel 7/Output
//     ModbusTask Outputs/GVL_Output.uniDO.stEbusDO.EL2889_09.DO8 <-> Channel 8/Output
//     ModbusTask Outputs/GVL_Output.uniDO.stEbusDO.EL2889_09.DO9 <-> Channel 9/Output
//   DAS_CoreSys/DAS_CoreSys Instance <-> Device 4 (EtherCAT) Allocate/Term 22 (EK1100)/Term 31 (EL2889)_10(Y2)
//     ModbusTask Outputs/GVL_Output.uniDO.stEbusDO.EL2889_10.DO{1..16} <-> Channel {1..16}/Output  (16 links)
//   DAS_CoreSys/DAS_CoreSys Instance <-> Device 4 (EtherCAT) Allocate/Term 22 (EK1100)/Term 33 (EL1889)_11(X4)
//     ModbusTask Inputs/GVL_Input.uniDI.stEbusDI.EL1889_11.DI{1..16} <-> Channel {1..16}/Input  (16 links)
//   DAS_CoreSys/DAS_CoreSys Instance <-> Device 6 (ECAT EIP Scanner (EL6652))
//     CoreSys Inputs/DAS_CoreSys.MachineControl.FanucRobot.List.ShippingRobot._FanucEIPState <-> Inputs/ECatState
//   DAS_CoreSys/DAS_CoreSys Instance <-> Device 6 (ECAT EIP Scanner (EL6652))/FANUC Robot R30iB+
//     CoreSys Inputs/DAS_CoreSys.MachineControl.FanucRobot.List.ShippingRobot._EIPConnectionState <-> Inputs/State
//     CoreSys Inputs/DAS_CoreSys.MachineControl.FanucRobot.List.ShippingRobot._rawIn_DI <-> DIO (Input/Output)/Inputs/noname0_arrBYTE
//     CoreSys Inputs/DAS_CoreSys.MachineControl.FanucRobot.List.ShippingRobot._rawIn_UI <-> UIO (Input/Output)/Inputs/noname0_arrBYTE
//     CoreSys Outputs/DAS_CoreSys.MachineControl.FanucRobot.List.ShippingRobot._rawOut_DO <-> DIO (Input/Output)/Outputs/noname0_arrBYTE
//     CoreSys Outputs/DAS_CoreSys.MachineControl.FanucRobot.List.ShippingRobot._rawOut_UO <-> UIO (Input/Output)/Outputs/noname0_arrBYTE
//   DAS_CoreSys/DAS_CoreSys Instance <-> Storage Fanuc Robot (ECAT EIP Scanner (EL6652))
//     CoreSys Inputs/DAS_CoreSys.MachineControl.FanucRobot.List.StorageRobot._FanucEIPState <-> Inputs/ECatState
//   DAS_CoreSys/DAS_CoreSys Instance <-> Storage Fanuc Robot (ECAT EIP Scanner (EL6652))/FANUC Robot R30iB+
//     CoreSys Inputs/DAS_CoreSys.MachineControl.FanucRobot.List.StorageRobot._EIPConnectionState <-> Inputs/State
//     CoreSys Inputs/DAS_CoreSys.MachineControl.FanucRobot.List.StorageRobot._rawIn_DI <-> DIO (Input/Output)/Inputs/noname0_arrBYTE
//     CoreSys Inputs/DAS_CoreSys.MachineControl.FanucRobot.List.StorageRobot._rawIn_UI <-> UIO (Input/Output)/Inputs/noname0_arrBYTE
//     CoreSys Outputs/DAS_CoreSys.MachineControl.FanucRobot.List.StorageRobot._rawOut_DO <-> DIO (Input/Output)/Outputs/noname0_arrBYTE
//     CoreSys Outputs/DAS_CoreSys.MachineControl.FanucRobot.List.StorageRobot._rawOut_UO <-> UIO (Input/Output)/Outputs/noname0_arrBYTE
//   DAS_CoreSys/DAS_CoreSys Instance <-> NC-Task 1 SAF/Axes/Axis 1|TurnTable
//     MotionSync Inputs/BATW.GVL_Motion.arAxisCtrl_gb[1].Admin.Axis.NcToPlc <-> Outputs/ToPlc
//     MotionSync Outputs/BATW.GVL_Motion.arAxisCtrl_gb[1].Admin.Axis.PlcToNc <-> Inputs/FromPlc
//   DAS_CoreSys/DAS_CoreSys Instance <-> NC-Task 1 SAF/Axes/Axis 2|RoundBelt
//     MotionSync Inputs/BATW.GVL_Motion.arAxisCtrl_gb[2].Admin.Axis.NcToPlc <-> Outputs/ToPlc
//     MotionSync Outputs/BATW.GVL_Motion.arAxisCtrl_gb[2].Admin.Axis.PlcToNc <-> Inputs/FromPlc
//   DAS_CoreSys/DAS_CoreSys Instance <-> NC-Task 1 SAF/Axes/Axis 3|AllocateRobot_X
//     MotionSync Inputs/BATW.GVL_Motion.arAxisCtrl_gb[3].Admin.Axis.NcToPlc <-> Outputs/ToPlc
//     MotionSync Outputs/BATW.GVL_Motion.arAxisCtrl_gb[3].Admin.Axis.PlcToNc <-> Inputs/FromPlc
//   DAS_CoreSys/DAS_CoreSys Instance <-> NC-Task 1 SAF/Axes/Axis 4|AllocateRobot_Y
//     MotionSync Inputs/BATW.GVL_Motion.arAxisCtrl_gb[4].Admin.Axis.NcToPlc <-> Outputs/ToPlc
//     MotionSync Outputs/BATW.GVL_Motion.arAxisCtrl_gb[4].Admin.Axis.PlcToNc <-> Inputs/FromPlc
//   DAS_CoreSys/DAS_CoreSys Instance <-> NC-Task 1 SAF/Axes/Axis 5|OutRobot_X
//     MotionSync Inputs/BATW.GVL_Motion.arAxisCtrl_gb[5].Admin.Axis.NcToPlc <-> Outputs/ToPlc
//     MotionSync Outputs/BATW.GVL_Motion.arAxisCtrl_gb[5].Admin.Axis.PlcToNc <-> Inputs/FromPlc
//   DAS_CoreSys/DAS_CoreSys Instance <-> NC-Task 1 SAF/Axes/Axis 6|OutRobot_Y
//     MotionSync Inputs/BATW.GVL_Motion.arAxisCtrl_gb[6].Admin.Axis.NcToPlc <-> Outputs/ToPlc
//     MotionSync Outputs/BATW.GVL_Motion.arAxisCtrl_gb[6].Admin.Axis.PlcToNc <-> Inputs/FromPlc
//   DAS_CoreSys/DAS_CoreSys Instance <-> NC-Task 1 SAF/Axes/Axis 7|RackMotor
//     MotionSync Inputs/BATW.GVL_Motion.arAxisCtrl_gb[7].Admin.Axis.NcToPlc <-> Outputs/ToPlc
//     MotionSync Outputs/BATW.GVL_Motion.arAxisCtrl_gb[7].Admin.Axis.PlcToNc <-> Inputs/FromPlc

CONFIGURATION DAS_CoreSys
    RESOURCE PLC ON TwinCAT3
        TASK ModbusTask(INTERVAL := T#5ms, PRIORITY := 21);
        PROGRAM ComModbusRTU WITH ModbusTask : ComModbusRTU;
        PROGRAM MAIN2_RS485 WITH ModbusTask : MAIN2_RS485;
    END_RESOURCE
END_CONFIGURATION

// ---- Library/00_PackML/02_Mode/E_UnitMode.TcDUT
{attribute 'qualified_only'}
TYPE E_UnitMode :
(
        Undefined   := 0, // Mode not defined.
        Auto        := 1, // Mode Auto, production...
        Mantainance := 2, // Mode Mantainance, repair or test...etc
        Manual      := 3, // Mode Manual, user manual control
        Homing      := 4 // Mode Homing, unit's home
)DINT;
END_TYPE

// ---- Library/10_Machine/12_MachineControl/DUTs/Cylinders/ST_CylinderList.TcDUT
TYPE
    ST_CylinderList :
    STRUCT
        fbUpCV_FeedInPress1             : FB_Cylinder;
        fbUpCV_FeedInPress2             : FB_Cylinder;
        fbUpCV_DiameterPress            : FB_Cylinder;
        fbUpCV_CamaraPress1             : FB_Cylinder;
        fbUpCV_CamaraPress2             : FB_Cylinder;
        fbUpCV_CamaraPress3             : FB_Cylinder;
        fbUpCV_CamaraPress4             : FB_Cylinder;
        fbUpCV_Block1                   : FB_Cylinder;
        fbUpCV_Block2                   : FB_Cylinder;
        fbUpCV_Block3                   : FB_Cylinder;
        fbUpCV_DiameterHoriz            : FB_Cylinder;
        fbUpCV_DiameterVert             : FB_Cylinder;
        fbUpCV_DiameterClamp            : FB_Cylinder;
        fbStackPush                     : FB_Cylinder;
        fbPullOutCV_AsidePress1         : FB_Cylinder;
        fbPullOutCV_AsidePress2         : FB_Cylinder;
        fbPullOutCV_AsideBlock          : FB_Cylinder;
        fbPullOutCV_BsidePress1         : FB_Cylinder;
        fbPullOutCV_BsidePress2         : FB_Cylinder;
        fbPullOutCV_BsideBlock          : FB_Cylinder;
        fbLowCV_Press1                  : FB_Cylinder;
        fbLowCV_Press2                  : FB_Cylinder;
        fbLowCV_Press3                  : FB_Cylinder;
        fbLowCV_Press4                  : FB_Cylinder;
        fbLowCV_Block1                  : FB_Cylinder;
        fbLowCV_Block2                  : FB_Cylinder;
        fbAllocateRobot_LeftVert1       : FB_Cylinder;
        fbAllocateRobot_LeftVert2       : FB_Cylinder;
        fbAllocateRobot_RightVert1      : FB_Cylinder;
        fbAllocateRobot_RightVert2      : FB_Cylinder;
        fbAllocateRobot_LeftClamp1      : FB_Cylinder;
        fbAllocateRobot_LeftClamp2      : FB_Cylinder;
        fbAllocateRobot_RightClamp1     : FB_Cylinder;
        fbAllocateRobot_RightClamp2     : FB_Cylinder;
        fbRoundBelt_WorkZone_Press      : FB_Cylinder;
        fbRoundBelt_WorkZone_Plug       : FB_Cylinder;
        fbRoundBelt_ChargeZone_Plug     : FB_Cylinder;
        fbRoundBelt_TransmitCVZone_Plug : FB_Cylinder;
        fbOutRobot_AsideVert            : FB_Cylinder;
        fbOutRobot_BsideVert            : FB_Cylinder;
        fbOutRobot_AsideClamp           : FB_Cylinder;
        fbOutRobot_BsideClamp           : FB_Cylinder;
        fbTransmitCV_CamaraHoriz        : FB_Cylinder;
        fbDifferentSizeCV_Press2        : FB_Cylinder;
        fbDifferentSizeCV_Press1        : FB_Cylinder;
        fbDifferentSizeCV_Block1        : FB_Cylinder;
        fbSameSizeCV_Press4             : FB_Cylinder;
        fbSameSizeCV_Press3             : FB_Cylinder;
        fbSameSizeCV_Press2             : FB_Cylinder;
        fbSameSizeCV_Press1             : FB_Cylinder;
        fbSameSizeCV_Block2             : FB_Cylinder;
        fbSameSizeCV_Block1             : FB_Cylinder;
        fbTurntable_Press               : FB_Cylinder;
		fbShippingBuffer_Press			: FB_Cylinder;		// Edited by Gamin 20260410 新增，空指向僅建立空殼防止編譯錯誤。
    END_STRUCT
END_TYPE

// ---- Library/10_Machine/12_MachineControl/DUTs/FanucRobot/ST_FanucRobotList.TcDUT
TYPE
    ST_FanucRobotList :
    STRUCT
        StorageRobot  : FB_FanucRobot_Basic_V2;
        ShippingRobot : FB_FanucRobot_Basic_V2;
    END_STRUCT
END_TYPE

// ---- Library/10_Machine/12_MachineControl/DUTs/FanucRobot/UNI_FanucRobotList.TcDUT
TYPE
    UNI_FanucRobotList :
    UNION
        arFanucRobot : ARRAY[1..2] OF FB_FanucRobot_Basic_V2;
        List         : ST_FanucRobotList;
    END_UNION
END_TYPE

// ---- Library/10_Machine/12_MachineControl/DUTs/Motor/ST_SameSizeCVRequest.TcDUT
// 同尺寸軌道仲裁 request struct (Phase 2 集中式 motor control)
// 各 sub-FB 只寫請求 flag,不直接操作 Motor.List.TransmitSameSideCV。
// 由 FB_MachineControl.A20_ConveyorArbitration 每 scan 仲裁,真正下 M_MoveBackward / M_MoveForward / M_MotorStop。
// 仲裁優先序:HoldStill > 方向衝突 (停) > Backward / Forward > 預設停。
TYPE
    ST_SameSizeCVRequest :
    STRUCT
        // ===== Backward 請求 (倒帶方向 — 送盒入倉 / 推走 / 入鏡頭) =====
        bScan_NeedBackward              : BOOL;     // FB_ShippingPlateScan Phase 2 放盒
        bShippingTransfer_NeedBackward  : BOOL;     // FB_ShippingRobotTransfer Put 到 TransmitCV_End
        bCamera_NeedBackward            : BOOL;     // FB_SameSizeCVCamera_Reverse 送盒到拍照位 / 離開
        bWareHouse_NeedBackward         : BOOL;     // FB_SameSizeCV_ReverseBoxToWareHouse Phase 1/3 送盒到 NearStorage

        // ===== Forward 請求 (極少用 — Get from TransmitCV_End 場景) =====
        bShippingTransfer_NeedForward   : BOOL;     // FB_ShippingRobotTransfer Get from TransmitCV_End

        // ===== HoldStill 請求 (強制停 — 對位 / 拍照 / 取盒) =====
        bCamera_HoldStill               : BOOL;     // 拍照時必須靜止
        bWareHouse_HoldStill            : BOOL;     // 大手臂取盒時必須靜止
    END_STRUCT
END_TYPE

// ---- Library/10_Machine/12_MachineControl/DUTs/Setup/ST_AxisPara.TcDUT
TYPE
    ST_AxisPara :
    STRUCT
        Manual   : ST_AxisPara_Manual; // In Manual mode, Axis control will use.
        HalfAuto : ST_AxisPara_HalfAuto; // In HalfAuto mode, Axis control will use.
        Auto     : ST_AxisPara_Auto; // In AutoMode, Axis control will use.
        Homing   : ST_AxisPara_Homing; // In HomingMode, Axis control will use.
    END_STRUCT
END_TYPE

// ---- Library/10_Machine/12_MachineControl/DUTs/Setup/ST_PositionTable.TcDUT
TYPE
    ST_PositionTable :
    STRUCT
        Zone  : STRING; // Object zone
        Index : INT; // The position index in the zone
        X_Pos : LREAL; // X-Axis target position (Unit: mm)
        Y_Pos : LREAL; // Y-Axis target position (Unit: mm)
        R_Pos : LREAL; // R-Axis target position (Unit: deg)
        Robot : INT; // unuse 
        Clip  : E_ClipNo; // Select Object clip no.
    END_STRUCT
END_TYPE

// ---- Library/10_Machine/12_MachineControl/DUTs/Setup/ST_SetupAxis.TcDUT
TYPE
    ST_SetupAxis :
    STRUCT
        TurnTable  : ST_AxisPara; // Setup TurnTable Axis parameter, in DAS_CoreSys
        RoundBelt  : ST_AxisPara; // Setup RoundBelt Axis parameter, in DAS_CoreSys
        OutRobot_X : ST_AxisPara; // Setup OutRobot_X Axis parameter, in DAS_CoreSys
        OutRobot_Y : ST_AxisPara; // Setup OutRobot_Y Axis parameter, in DAS_CoreSys
        Allocate_X : ST_AxisPara; // Setup Allocate_X Axis parameter, in DAS_CoreSys
        Allocate_Y : ST_AxisPara; // Setup Allocate_Y Axis parameter, in DAS_CoreSys
		RackMotor  : ST_AxisPara; // Setup RackMotor  Axis parameter, in DAS_CoreSys
    END_STRUCT
END_TYPE

// ---- Library/10_Machine/12_MachineControl/DUTs/Setup/ST_SetupFanucRobot.TcDUT
TYPE
    ST_SetupFanucRobot :
    STRUCT
        RobotVelocity : LREAL :=20 ;
		ZoneCCD : ST_FanucRobotCCDSetting;
    END_STRUCT
END_TYPE

// ---- Library/10_Machine/12_MachineControl/DUTs/Setup/ST_SetupMotor.TcDUT
TYPE
    ST_SetupMotor :
    STRUCT
        WareHouseCV_10          : ST_MotorPara;
        WareHouseCV_09          : ST_MotorPara;
        WareHouseCV_08          : ST_MotorPara;
        WareHouseCV_07          : ST_MotorPara;
        WareHouseCV_06          : ST_MotorPara;
        WareHouseCV_05          : ST_MotorPara;
        WareHouseCV_04          : ST_MotorPara;
        WareHouseCV_03          : ST_MotorPara;
        WareHouseCV_02          : ST_MotorPara;
        WareHouseCV_01          : ST_MotorPara;
        WareHouseCV_20          : ST_MotorPara;
        WareHouseCV_19          : ST_MotorPara;
        WareHouseCV_18          : ST_MotorPara;
        WareHouseCV_17          : ST_MotorPara;
        WareHouseCV_16          : ST_MotorPara;
        WareHouseCV_15          : ST_MotorPara;
        WareHouseCV_14          : ST_MotorPara;
        WareHouseCV_13          : ST_MotorPara;
        WareHouseCV_12          : ST_MotorPara;
        WareHouseCV_11          : ST_MotorPara;
        UpCV                    : ST_MotorPara;
        LowCV                   : ST_MotorPara;
        PullOutCV_A             : ST_MotorPara;
        PullOutCV_B             : ST_MotorPara;
        TransmitSameSideCV      : ST_MotorPara;
        TransmitDifferentSideCV : ST_MotorPara;
    END_STRUCT
END_TYPE

// ---- Library/10_Machine/12_MachineControl/DUTs/Setup/ST_SetupPara.TcDUT
TYPE
    ST_SetupPara :
    STRUCT
        Cylinders     : ST_SetupCylinder;
        Axes          : ST_SetupAxis;
        Motor         : ST_SetupMotor;
        PositionTable : ARRAY[1..200] OF ST_PositionTable;
        StorageRobot  : ST_SetupFanucRobot;
        ShippingRobot : ST_SetupFanucRobot;
        Mechanical    : ST_Setup_Mechanical;
		Light 		  : ST_Setup_Light;
		ShippingRobot_DockTestSignal : BOOL;
    END_STRUCT
END_TYPE

// ---- Library/10_Machine/12_MachineControl/DUTs/Setup/ST_Setup_Light.TcDUT
TYPE
    ST_Setup_Light :
    STRUCT
        Storage_EleBoxLight_Off : BOOL; // True : Turn off light
        Storage_AreaLight_Off : BOOL; // True : Turn off light
        Allocated_AreaLight_Off : BOOL; //True : Turn off light
    END_STRUCT
END_TYPE

// ---- Library/10_Machine/12_MachineControl/DUTs/Setup/ST_Setup_Mechanical.TcDUT
TYPE
    ST_Setup_Mechanical :
    STRUCT
        //配針手臂在圓帶的盒的左右的間距
        Allocate_box_leftandRight_Distance : LREAL;
        //配針手臂在圓帶的盒的上下的間距
        Allocate_box_UpandDown_Distance : LREAL;  
		// timeout setting
		stTimeoutSetting	:st_ServiceTimeoutSetting;
		// RS485 by pass
		stModbusByPass			:st_ModbusSwitchOff;
		//SafetyDoor
		stSafetyByPass			:st_SafetyByPass;
    END_STRUCT
END_TYPE

// ---- Library/10_Machine/18_HMI_Handshake/DUTs/Allocated/ST_HMI_AllocateArea.TcDUT
TYPE
    ST_HMI_AllocateArea :
    STRUCT
        Manual   : ST_Manual_Allocated;   // Allocated manual control
        HalfAuto : ST_HalfAuto_Allocated; // Allocated half-auto contorl
        //Auto     : ST_Auto_Allocated;     // Allocated auto control
    END_STRUCT
END_TYPE

// ---- Library/10_Machine/18_HMI_Handshake/DUTs/Allocated/ST_Manual_Allocated.TcDUT
TYPE
    ST_Manual_Allocated :
    STRUCT
        OutRobot       : ST_Manual_OutRobot;       // Allocated out robot manual control
        AllocatedRobot : ST_Manual_AllocatedRobot; // Allocated allocated robot manual control
        RoundBelt      : ST_Manual_RoundBelt;      // Allocated round belt manual control
        TurnTable      : ST_Manual_TurnTable;      // Allocated turn table manual control
        PullOutCV      : ST_Manual_PullOut;        // Allocated pullout conveyor manual control
        TransCV        : ST_Manual_TransCV;        // Allocated transmit conveyor manual control
    END_STRUCT
END_TYPE

// ---- Library/10_Machine/18_HMI_Handshake/DUTs/Allocated/ST_Manual_AllocatedRobot.TcDUT
TYPE
    ST_Manual_AllocatedRobot :
    STRUCT
        LeftVert1   : ST_SignleValve; // AllocateRobot LeftVert1 cylinder controll
        LeftVert2   : ST_SignleValve; // AllocateRobot LeftVert2 cylinder controll
        RightVert1  : ST_SignleValve; // AllocateRobot RightVert1 cylinder controll
        RightVert2  : ST_SignleValve; // AllocateRobot RightVert2 cylinder controll
        LeftClamp1  : ST_SignleValve; // AllocateRobot LeftClamp1 cylinder controll
        LeftClamp2  : ST_SignleValve; // AllocateRobot LeftClamp2 cylinder controll
        RightClamp1 : ST_SignleValve; // AllocateRobot RightClamp1 cylinder controll
        RightClamp2 : ST_SignleValve; // AllocateRobot RightClamp2 cylinder controll
        AxisX       : ST_Manual_Axis; // AllocateRobot AxisX controll
        AxisY       : ST_Manual_Axis; // AllocateRobot AxisY controll
    END_STRUCT
END_TYPE

// ---- Library/10_Machine/18_HMI_Handshake/DUTs/Allocated/ST_Manual_Axis.TcDUT
TYPE ST_Manual_Axis :
STRUCT
	JOG : ST_AXIS_JOG;
	PTP : ST_AXIS_PTP;
	Homing : ST_AXIS_HOMING;
END_STRUCT
END_TYPE

// ---- Library/10_Machine/18_HMI_Handshake/DUTs/Allocated/ST_Manual_PullOut.TcDUT
TYPE
    ST_Manual_PullOut :
    STRUCT
        AsidePress1 : ST_SignleValve;
        AsidePress2 : ST_SignleValve;
        AsideBlock  : ST_SignleValve;
        BsidePress1 : ST_SignleValve;
        BsidePress2 : ST_SignleValve;
        BsideBlock  : ST_SignleValve;
        PullOutCV_A : ST_MotorCommand;
        PullOutCV_B : ST_MotorCommand;
    END_STRUCT
END_TYPE

// ---- Library/10_Machine/18_HMI_Handshake/DUTs/Allocated/ST_Manual_RoundBelt.TcDUT
TYPE
    ST_Manual_RoundBelt :
    STRUCT
        WorkZone_Press      : ST_SignleValve;
        WorkZone_Plug       : ST_SignleValve;
        ChargeZone_Plug     : ST_SignleValve;
        TransmitCVZone_Plug : ST_SignleValve;
        Axis                : ST_Manual_Axis; // RoundBelt Axis controll

    END_STRUCT
END_TYPE

// ---- Library/10_Machine/18_HMI_Handshake/DUTs/Allocated/ST_Manual_TransCV.TcDUT
TYPE
    ST_Manual_TransCV :
    STRUCT
        CamaraHoriz             : ST_SignleValve;
        DifferentSizeCV_Press2  : ST_SignleValve;
        DifferentSizeCV_Press1  : ST_SignleValve;
        DifferentSizeCV_Block1  : ST_SignleValve;
        SameSizeCV_Press4       : ST_SignleValve;
        SameSizeCV_Press3       : ST_SignleValve;
        SameSizeCV_Press2       : ST_SignleValve;
        SameSizeCV_Press1       : ST_SignleValve;
        SameSizeCV_Block2       : ST_SignleValve;
        SameSizeCV_Block1       : ST_SignleValve;
        TransmitSameSideCV      : ST_MotorCommand;
        TransmitDifferentSideCV : ST_MotorCommand;
    END_STRUCT
END_TYPE

// ---- Library/10_Machine/18_HMI_Handshake/DUTs/E_AllocationJob.TcDUT
{attribute 'qualified_only'}
{attribute 'strict'}
TYPE E_AllocationJob :
(	PreDataProcess:=-1,
	Idle:=0,	
	Initial ,	
	CheckRotateBeltStation,
	MovingRotateBeltStation,
	MovedRotateBeltStation,
	CheckRotateBeltStation_SimpleAllocatePlacing,
	MovingRotateBeltStation_SimpleAllocatePlacing,
	MovedRotateBeltStation_SimpleAllocatePlacing,
	CheckBoxReadyOnAllocatePosOfRoundBelt,
	CheckBoxReadyOnRoundBelt_SimpleAllocateMode,
	MoveToTargetPos,
	MovingToTargetPos,
	CylinderDownPick,
	ClipColse,	
	CylinderUpPick,
	MoveToPlacingPos,
	MovingToPlacingPos,
	CylinderDownPlace,
	ClipOpen,		
	CylinderUpPlace,
	CheckNeedlePlaced,
	Defult,
	Finish,
	Error,
	CheckNeedlePick,
	CheckNeedlePlace,
	IfNextPTP_Picking,
	IfNextPTP_Placing,
	CheckBoxesOnTurnTableReady,
	FinalCleanup		// 最後一筆完成後的硬體歸位 gate (cylinders/clips/Press 全縮回 + RoundBelt idle 才允許 _Executed)

);
END_TYPE

// ---- Library/10_Machine/18_HMI_Handshake/DUTs/IOMonitor/ST_HMI_IOMonitor.TcDUT
TYPE
    ST_HMI_IOMonitor :
    STRUCT
        Input  : ST_InputTable_MitsubishiWithWheelHouse;
        Output : ST_OutputTable_Mitsubishi;
		
    END_STRUCT
END_TYPE

// ---- Library/10_Machine/18_HMI_Handshake/DUTs/IOMonitor/ST_InputTable_MitsubishiWithWheelHouse.TcDUT
TYPE ST_InputTable_MitsubishiWithWheelHouse EXTENDS ST_InputTable_Mitsubishi :
STRUCT
	arWheelhouseInput : ARRAY[1..400] OF BOOL;
END_STRUCT
END_TYPE

// ---- Library/10_Machine/18_HMI_Handshake/DUTs/Shipping/ST_HMI_ShippingArea.TcDUT
TYPE
    ST_HMI_ShippingArea :
    STRUCT
        Manual   : ST_Manual_Shipping;
        //HalfAuto : ST_HalfAuto_Shipping;
        //Auto     : ST_Auto_Shipping;
    END_STRUCT
END_TYPE

// ---- Library/10_Machine/18_HMI_Handshake/DUTs/Status/ST_AXES_STATUS.TcDUT
TYPE ST_AXES_STATUS :
    STRUCT
        TurnTable       : ST_SINGLEAXIS_STATUS; // TurnTable Axis status
        RoundBelt       : ST_SINGLEAXIS_STATUS; // RoundBelt Axis status
        Allocate_X      : ST_SINGLEAXIS_STATUS; // AllocateRRobot AxisX status
        Allocate_Y      : ST_SINGLEAXIS_STATUS; // AllocateRobot AxisY status
        OutRobot_X      : ST_SINGLEAXIS_STATUS; // OutRobot AxisX status
        OutRobot_Y      : ST_SINGLEAXIS_STATUS; // OutRobot AxisY status
		RackMotor : ST_SINGLEAXIS_STATUS; // Rack motor status
    END_STRUCT
END_TYPE

// ---- Library/10_Machine/18_HMI_Handshake/DUTs/Status/ST_HMI_MachineStatus.TcDUT
TYPE
    ST_HMI_MachineStatus :
    STRUCT
        Manual    : ST_Manual_Status;
        //HalfAuto  : ST_HalfAuto_Status;
        //Auto      : ST_Auto_Status;
        Axes      : ST_AXES_STATUS;
        Cylinders : ST_CylinderStatus;
        Motor     : ST_MotorStatus;
    END_STRUCT
END_TYPE

// ---- Library/10_Machine/18_HMI_Handshake/DUTs/Storage/ST_HMI_StorageArea.TcDUT
TYPE
    ST_HMI_StorageArea :
    STRUCT
        Manual   : ST_Manual_Storage;
        //HalfAuto : ST_HalfAuto_Storage;	//裡面空白結構會導致c# 交握Size出問題
        //Auto     : ST_Auto_Storage;
    END_STRUCT
END_TYPE

// ---- Library/10_Machine/18_HMI_Handshake/DUTs/Storage/ST_Manual_FanucRobot.TcDUT
TYPE ST_Manual_FanucRobot :
STRUCT
	//============================   Command  ==================================
	ClampA_Open  : BOOL; // FncRobotCommand : True: set clampA open 
	ClampA_Close : BOOL; // FncRobotCommand : True: Set ClampA Close
	ClampB_Open  : BOOL; // FncRobotCommand : True: Set ClampB Open
	ClampB_Close : BOOL; // FncRobotCommand : True: Set ClampB Close
	ByPassClampSensor : BOOL; // FncRobotCommand : True : Bypass clampA and clampB
	
	//FanucRobot Area Laser Function
	bStorageA_LaserSwitch	: BOOL := TRUE;
	bStorageB_LaserSwitch	: BOOL := TRUE;
	bRoundBelt_LaserSwitch	: BOOL ;
	bPrep_LaserSwitch		: BOOL := TRUE;
	bNeedle_LaserSwitch		: BOOL := TRUE;
	bConveyor_LaserSwitch	: BOOL := TRUE;
	bRemoval_LaserSwitch	: BOOL := TRUE;
	
	//Fanuc Robot Vision Function
	bRoundBelt_Vision_Switch	: BOOL;
	bPrep_Vision_Switch			: BOOL;
	bNeedle_Vision_Switch		: BOOL;
	bRemoval_Vision_Switch		: BOOL;
	//==========================================================================
	
	// ============================  Status  ===================================
	ClampA_Open_Status 		: BOOL;   // FncRobotStatus : True : ClampA open
    ClampB_Open_Status 		: BOOL;   // FncRobotStatus : True : ClampB open
    ClampA_SensorStatus 	: BOOL;   // FncRobotStatus : True : ClampA sensor detact
    ClampB_SensorStatus 	: BOOL;   // FncRobotStatus : True : CLampB sensor detact
	
	bStorageA_LaserStatus	: BOOL;
	bStorageB_LaserStatus	: BOOL;
	bRoundBelt_LaserStatus	: BOOL;
	bPrep_LaserStatus		: BOOL;
	bNeedle_LaserStatus		: BOOL;
	bConveyor_LaserStatus	: BOOL;
	bRemoval_LaserStatus	: BOOL;
	
	ClampA1_Laser_Status	: BOOL;
	ClampB1_Laser_Status	: BOOL;
	ClampA2_Laser_Status	: BOOL;
	ClampB2_Laser_Status	: BOOL;
	
	bRoundBelt_Vision_Status	: BOOL;
	bPrep_Vision_Status			: BOOL;
	bNeedle_Vision_Status		: BOOL;
	bRemoval_Vision_Status		: BOOL;
	//==========================================================================
	
END_STRUCT
END_TYPE

// ---- Library/10_Machine/18_HMI_Handshake/OLD_DUTs/E_FeedInToWareHouse_PlaceArea.TcDUT
{attribute 'qualified_only'}
{attribute 'strict'}
TYPE
    E_FeedInToWareHouse_PlaceArea :
    (
        Undefined := 0,
        WareHouseA := 1,
        WareHouseB := 2,
        PullOutOuter := 3,  // PullOutConveyor I4_Slide (右側,面對操作員 / 機台外側)
        PullOutInner := 4   // PullOutConveyor I3_Slide (左側,面對操作員 / 機台內側)
    )UINT;
END_TYPE

// ---- Library/10_Machine/18_HMI_Handshake/OLD_DUTs/ST_AutoMode_FeedInToWareHouseBox.TcDUT
TYPE ST_AutoMode_FeedInToWareHouseBox :
STRUCT
	Command 		: ST_FeedInToWareHouse_Ctrl;
	Status 			: ST_FeedInToWareHouse_Status;
	Info 			: ST_FeedInToWareHouseBox_Info;
	AClampMoveDone	: BOOL;
	BClampMoveDone	: BOOL;
END_STRUCT
END_TYPE

// ---- Library/10_Machine/18_HMI_Handshake/OLD_DUTs/ST_AutoMode_RobotSelfHoming.TcDUT
TYPE ST_AutoMode_RobotSelfHoming :
STRUCT
	Command	: ST_CommandBasic;
	Status	: ST_StatusBasic;
	BypassFeedOutToNGCV	: BOOL;
END_STRUCT
END_TYPE

// ---- Library/10_Machine/18_HMI_Handshake/OLD_DUTs/ST_AutoMode_ShippingLeftSideTransCV.TcDUT
TYPE ST_AutoMode_ShippingLeftSideTransCV :
STRUCT
	Command : ST_CommandBasic;
	Status	: ST_StatusBasic;
	ShippingTransCVRequest_LeftSide : BOOL;		//C# to PLC
END_STRUCT
END_TYPE

// ---- Library/10_Machine/18_HMI_Handshake/OLD_DUTs/DataCore/st_ADS_X.TcDUT
TYPE st_ADS_X :
STRUCT
	
X0 : ARRAY [0..15] OF BOOL;
X1 : ARRAY [0..15] OF BOOL;
X2 : ARRAY [0..15] OF BOOL;
X3 : ARRAY [0..15] OF BOOL;
X4 : ARRAY [0..15] OF BOOL;
X5 : ARRAY [0..15] OF BOOL;
X6 : ARRAY [0..15] OF BOOL;
X7 : ARRAY [0..15] OF BOOL; 
X8 : ARRAY [0..15] OF BOOL; 
X9 : ARRAY [0..15] OF BOOL; 
X10 : ARRAY [0..15] OF BOOL; 

 
D0 : ARRAY [0..15] OF LREAL;
M2 : ARRAY [0..399] OF BOOL;

//Runs : ARRAY[1..12] OF BOOL;

END_STRUCT
END_TYPE

// ---- Library/10_Machine/18_HMI_Handshake/OLD_DUTs/DataCore/st_ADS_Y.TcDUT
TYPE st_ADS_Y :
STRUCT

Y0 : ARRAY [0..15] OF BOOL;
Y1 : ARRAY [0..15] OF BOOL;
Y2 : ARRAY [0..15] OF BOOL;
Y3 : ARRAY [0..15] OF BOOL;
Y4 : ARRAY [0..15] OF BOOL;
Y5 : ARRAY [0..15] OF BOOL;
Y6 : ARRAY [0..15] OF BOOL;
Y7 : ARRAY [0..15] OF BOOL;
Y8 : ARRAY [0..15] OF BOOL;	
Y9 : ARRAY [0..15] OF BOOL;	
Y10 : ARRAY [0..15] OF BOOL;	

M0 : ARRAY [0..95] OF BOOL;
M1 : ARRAY [0..141] OF BOOL;

D0 : ARRAY [0..95] OF LREAL;
D1 : ARRAY [0..95] OF LREAL;
END_STRUCT
END_TYPE

// ---- Library/10_Machine/18_HMI_Handshake/OLD_DUTs/E_ClampWork.TcDUT
{attribute 'qualified_only'}
{attribute 'strict'}
TYPE E_ClampWork :
(
	Undefined := 0,
	NoWork := 1,
	Work := 2
);
END_TYPE

// ---- Library/10_Machine/18_HMI_Handshake/OLD_DUTs/E_FeedInEmptyBox_PickUpArea.TcDUT
{attribute 'qualified_only'}
{attribute 'strict'}
TYPE
    E_FeedInEmptyBox_PickUpArea :
    (
        Undefined := 0,
        WareHouseA := 1,
        WareHouseB := 2,
		PullOutConveyor := 3
    ) UINT;
END_TYPE

// ---- Library/10_Machine/18_HMI_Handshake/OLD_DUTs/E_FeedInEmptyBox_PlaceArea.TcDUT
{attribute 'qualified_only'}
TYPE
    E_FeedInEmptyBox_PlaceArea :
    (
        Undefine := 0,	// No Setting
        SameSizeConveyor := 1, // Target is allocate FeedIn conveyor same size side.
        DiffSizeConveyor := 2 // Target is allocate FeedIn conveyor different size side.
    ) UINT;
END_TYPE

// ---- Library/10_Machine/18_HMI_Handshake/OLD_DUTs/E_HoleIndex_X.TcDUT
{attribute 'qualified_only'}
TYPE E_HoleIndex_X :
(
    Row1 :=1,
    Row2,
    Row3,
    Row4,
    Row5,
    Row6,
    Row7,
    Row8,
    Row9,
    Row10
);
END_TYPE

// ---- Library/10_Machine/18_HMI_Handshake/OLD_DUTs/E_HoleIndex_Y.TcDUT
{attribute 'qualified_only'}
TYPE E_HoleIndex_Y :
(
    Column1 :=1,
    Column2,
    Column3,
    Column4,
    Column5
);
END_TYPE

// ---- Library/10_Machine/18_HMI_Handshake/OLD_DUTs/E_MachineMode.TcDUT
TYPE E_MachineMode :
(
	UNDEFINE := 0,
	MANUAL	:=1		  ,
	AUTO	:=2		  ,
	SERVICE :=3,
	ModeSelect:=99
)INT;
END_TYPE

// ---- Library/10_Machine/18_HMI_Handshake/OLD_DUTs/E_MachineState.TcDUT
{attribute 'qualified_only'}
{attribute 'strict'}
TYPE E_MachineState :
(
	Default := 0,
	NotHomed,
	Homing,
	Homed,
	Starting,
	Stopping,
	Running,
	StandBy,
	Error
);
END_TYPE

// ---- Library/10_Machine/18_HMI_Handshake/OLD_DUTs/E_PullOutConveyorAddress.TcDUT
{attribute 'qualified_only'}
{attribute 'strict'}
TYPE E_PullOutConveyorAddress :
(
	Undefined := 0,
	I3_Slide, 	// it's left slide of face machine operating side 
	I4_Slide	// it's right slide of face machine operating side 
);
END_TYPE

